C07321=1112.756,31.841,-53.401,179.866,6.990,149.335
C07322=1112.751,32.090,-53.417,179.867,6.994,149.335
C07323=1112.747,32.340,-53.432,179.868,6.998,149.336
C07324=1112.742,32.589,-53.448,179.869,7.003,149.337
C07325=1112.736,32.839,-53.464,179.870,7.007,149.337
C07326=1112.731,33.089,-53.480,179.870,7.011,149.338
C07327=1112.727,33.338,-53.495,179.871,7.015,149.339
C07328=1112.722,33.587,-53.511,179.872,7.020,149.339
C07329=1112.717,33.837,-53.527,179.874,7.024,149.340
C07330=1112.711,34.086,-53.542,179.875,7.028,149.341
C07331=1112.706,34.336,-53.558,179.875,7.032,149.341
C07332=1112.702,34.585,-53.573,179.876,7.036,149.342
C07333=1112.697,34.834,-53.590,179.877,7.040,149.343
C07334=1112.692,35.084,-53.605,179.878,7.045,149.343
C07335=1112.687,35.334,-53.621,179.879,7.049,149.344
C07336=1112.681,35.583,-53.637,179.880,7.053,149.345
C07337=1112.676,35.832,-53.653,179.881,7.057,149.345
C07338=1112.672,36.046,-53.667,179.882,7.061,149.346
C07339=1112.668,36.260,-53.680,179.883,7.064,149.346
C07340=1112.664,36.475,-53.693,179.884,7.067,149.347
C07341=1112.660,36.690,-53.707,179.884,7.071,149.348
C07342=1112.655,36.904,-53.720,179.885,7.075,149.348
C07343=1112.651,37.118,-53.734,179.886,7.078,149.349
C07344=1112.647,37.332,-53.748,179.887,7.082,149.349
C07345=1112.642,37.547,-53.761,179.888,7.086,149.350
C07346=1112.637,37.796,-53.778,179.889,7.089,149.350
C07347=1112.633,38.046,-53.794,179.890,7.094,149.351
C07348=1112.627,38.294,-53.810,179.891,7.098,149.352
C07349=1112.622,38.544,-53.826,179.892,7.102,149.352
C07350=1112.617,38.794,-53.842,179.893,7.107,149.353
C07351=1112.612,39.043,-53.858,179.893,7.110,149.354
C07352=1112.607,39.293,-53.874,179.895,7.114,149.354
C07353=1112.602,39.542,-53.890,179.896,7.118,149.355
C07354=1112.598,39.792,-53.906,179.897,7.123,149.355
C07355=1112.592,40.041,-53.922,179.898,7.127,149.356
C07356=1112.588,40.290,-53.938,179.899,7.130,149.357
C07357=1112.583,40.540,-53.953,179.900,7.135,149.357
C07358=1112.578,40.789,-53.970,179.901,7.139,149.358
C07359=1112.573,41.039,-53.986,179.902,7.143,149.359
C07360=1112.568,41.287,-54.002,179.903,7.147,149.359
C07361=1112.563,41.538,-54.018,179.904,7.152,149.360
C07362=1112.557,41.787,-54.035,179.905,7.155,149.360
C07363=1112.553,42.037,-54.051,179.906,7.159,149.361
C07364=1112.548,42.285,-54.067,179.907,7.164,149.362
C07365=1112.543,42.536,-54.083,179.908,7.168,149.362
C07366=1112.538,42.784,-54.099,179.910,7.172,149.363
C07367=1112.533,43.034,-54.115,179.910,7.175,149.363
C07368=1112.528,43.283,-54.131,179.911,7.180,149.364
C07369=1112.523,43.533,-54.147,179.912,7.184,149.365
C07370=1112.518,43.782,-54.164,179.913,7.188,149.365
C07371=1112.514,44.032,-54.180,179.915,7.192,149.366
C07372=1112.508,44.281,-54.196,179.915,7.196,149.366
C07373=1112.504,44.531,-54.213,179.916,7.200,149.367
C07374=1112.499,44.779,-54.229,179.917,7.204,149.368
C07375=1112.494,45.029,-54.245,179.919,7.208,149.368
C07376=1112.489,45.278,-54.261,179.920,7.213,149.369
C07377=1112.483,45.529,-54.278,179.921,7.217,149.369
C07378=1112.479,45.778,-54.294,179.922,7.220,149.370
C07379=1112.474,46.027,-54.311,179.923,7.224,149.371
C07380=1112.469,46.277,-54.327,179.924,7.229,149.371
C07381=1112.464,46.526,-54.343,179.925,7.233,149.372
C07382=1112.459,46.775,-54.360,179.927,7.237,149.372
C07383=1112.454,47.024,-54.376,179.927,7.240,149.373
C07384=1112.449,47.274,-54.393,179.928,7.245,149.374
C07385=1112.444,47.524,-54.409,179.929,7.249,149.374
C07386=1112.439,47.773,-54.425,179.931,7.253,149.375
C07387=1112.435,48.022,-54.442,179.932,7.257,149.375
C07388=1112.429,48.272,-54.458,179.933,7.261,149.376
C07389=1112.424,48.521,-54.475,179.934,7.265,149.376
C07390=1112.420,48.771,-54.492,179.935,7.269,149.377
C07391=1112.414,49.020,-54.508,179.936,7.273,149.378
C07392=1112.410,49.269,-54.525,179.938,7.277,149.378
C07393=1112.405,49.519,-54.540,179.939,7.281,149.379
C07394=1112.400,49.733,-54.556,179.940,7.284,149.379
C07395=1112.396,49.948,-54.569,179.940,7.288,149.380
C07396=1112.392,50.161,-54.584,179.942,7.292,149.380
C07397=1112.388,50.376,-54.597,179.943,7.295,149.381
C07398=1112.384,50.589,-54.612,179.944,7.298,149.381
C07399=1112.379,50.804,-54.626,179.944,7.302,149.382
C07400=1112.375,51.018,-54.641,179.946,7.306,149.382
C07401=1112.371,51.233,-54.655,179.947,7.309,149.383
C07402=1112.366,51.481,-54.671,179.948,7.313,149.383
C07403=1112.361,51.731,-54.688,179.949,7.317,149.384
C07404=1112.356,51.981,-54.705,179.950,7.320,149.384
C07405=1112.351,52.230,-54.721,179.951,7.325,149.385
C07406=1112.346,52.479,-54.738,179.952,7.329,149.386
C07407=1112.342,52.729,-54.755,179.954,7.333,149.386
C07408=1112.337,52.978,-54.771,179.955,7.337,149.387
C07409=1112.331,53.227,-54.789,179.956,7.341,149.387
C07410=1112.327,53.477,-54.805,179.957,7.344,149.388
C07411=1112.322,53.726,-54.822,179.958,7.349,149.388
C07412=1112.317,53.975,-54.839,179.959,7.353,149.389
C07413=1112.312,54.225,-54.856,179.961,7.357,149.389
C07414=1112.306,54.474,-54.873,179.962,7.361,149.390
C07415=1112.302,54.724,-54.889,179.964,7.365,149.391
C07416=1112.297,54.973,-54.906,179.964,7.368,149.391
C07417=1112.292,55.223,-54.923,179.966,7.372,149.392
C07418=1112.287,55.472,-54.939,179.967,7.377,149.392
C07419=1112.282,55.721,-54.957,179.968,7.381,149.393
C07420=1112.277,55.971,-54.973,179.969,7.385,149.393
C07421=1112.272,56.220,-54.990,179.970,7.389,149.394
C07422=1112.267,56.469,-55.007,179.971,7.392,149.394
C07423=1112.263,56.719,-55.024,179.972,7.397,149.395
C07424=1112.257,56.969,-55.041,179.974,7.401,149.396
C07425=1112.253,57.217,-55.058,179.975,7.405,149.396
C07426=1112.247,57.467,-55.075,179.977,7.409,149.397
C07427=1112.243,57.716,-55.092,179.978,7.413,149.397
C07428=1112.238,57.966,-55.109,179.979,7.416,149.398
C07429=1112.233,58.215,-55.126,179.980,7.420,149.398
C07430=1112.227,58.465,-55.143,179.981,7.424,149.399
C07431=1112.223,58.713,-55.160,179.982,7.429,149.399
C07432=1112.218,58.963,-55.177,179.984,7.433,149.400
C07433=1112.213,59.213,-55.194,179.985,7.437,149.400
C07434=1112.208,59.462,-55.211,179.987,7.441,149.401
C07435=1112.203,59.711,-55.228,179.988,7.444,149.401
C07436=1112.198,59.960,-55.246,179.989,7.448,149.402
C07437=1112.194,60.210,-55.262,179.990,7.452,149.402
C07438=1112.189,60.460,-55.279,179.991,7.456,149.403
C07439=1112.184,60.709,-55.297,179.993,7.460,149.404
C07440=1112.179,60.958,-55.314,179.994,7.465,149.404
C07441=1112.174,61.207,-55.330,179.995,7.468,149.405
C07442=1112.169,61.456,-55.348,179.996,7.472,149.405
C07443=1112.164,61.706,-55.366,179.998,7.476,149.406
C07444=1112.159,61.956,-55.382,179.999,7.480,149.406
C07445=1112.155,62.205,-55.400,-180.000,7.484,149.407
C07446=1112.150,62.454,-55.417,-179.998,7.488,149.407
C07447=1112.145,62.704,-55.434,-179.997,7.492,149.408
C07448=1112.139,62.953,-55.452,-179.996,7.495,149.408
C07449=1112.135,63.202,-55.469,-179.995,7.500,149.409
C07450=1112.131,63.417,-55.484,-179.993,7.504,149.409
C07451=1112.127,63.630,-55.498,-179.993,7.507,149.410
C07452=1112.122,63.844,-55.513,-179.992,7.510,149.410
C07453=1112.119,64.059,-55.528,-179.990,7.514,149.411
C07454=1112.114,64.273,-55.543,-179.989,7.517,149.411
C07455=1112.109,64.487,-55.558,-179.988,7.520,149.412
C07456=1112.106,64.701,-55.573,-179.987,7.524,149.412
C07457=1112.101,64.915,-55.588,-179.986,7.527,149.412
C07458=1112.097,65.164,-55.605,-179.984,7.531,149.413
C07459=1112.092,65.414,-55.623,-179.983,7.535,149.413
C07460=1112.087,65.663,-55.641,-179.981,7.539,149.414
C07461=1112.082,65.913,-55.657,-179.981,7.543,149.415
C07462=1112.077,66.162,-55.675,-179.979,7.547,149.415
C07463=1112.072,66.412,-55.693,-179.978,7.550,149.415
C07464=1112.067,66.660,-55.710,-179.977,7.555,149.416
C07465=1112.062,66.910,-55.727,-179.975,7.559,149.417
C07466=1112.057,67.159,-55.745,-179.974,7.563,149.417
C07467=1112.052,67.409,-55.762,-179.972,7.567,149.418
C07468=1112.048,67.657,-55.779,-179.971,7.571,149.418
C07469=1112.043,67.907,-55.797,-179.970,7.574,149.419
C07470=1112.038,68.156,-55.815,-179.969,7.578,149.419
C07471=1112.033,68.406,-55.833,-179.967,7.582,149.420
C07472=1112.028,68.655,-55.850,-179.966,7.586,149.420
C07473=1112.023,68.904,-55.867,-179.964,7.590,149.421
C07474=1112.018,69.153,-55.885,-179.963,7.594,149.421
C07475=1112.013,69.403,-55.903,-179.962,7.598,149.422
C07476=1112.008,69.652,-55.921,-179.960,7.602,149.422
C07477=1112.003,69.902,-55.938,-179.959,7.606,149.423
C07478=1111.999,70.151,-55.955,-179.958,7.610,149.423
C07479=1111.994,70.400,-55.973,-179.957,7.614,149.424
C07480=1111.989,70.649,-55.991,-179.955,7.618,149.424
C07481=1111.984,70.899,-56.008,-179.954,7.622,149.425
C07482=1111.979,71.148,-56.026,-179.952,7.626,149.425
C07483=1111.974,71.397,-56.044,-179.951,7.630,149.426
C07484=1111.969,71.647,-56.062,-179.949,7.634,149.426
C07485=1111.965,71.896,-56.079,-179.948,7.638,149.427
C07486=1111.960,72.146,-56.097,-179.947,7.642,149.427
C07487=1111.955,72.395,-56.115,-179.945,7.646,149.428
C07488=1111.951,72.644,-56.133,-179.944,7.649,149.428
C07489=1111.945,72.894,-56.151,-179.943,7.653,149.429
C07490=1111.940,73.143,-56.169,-179.941,7.657,149.429
C07491=1111.936,73.393,-56.187,-179.940,7.661,149.430
C07492=1111.931,73.642,-56.205,-179.939,7.665,149.430
C07493=1111.926,73.891,-56.222,-179.937,7.669,149.431
C07494=1111.921,74.140,-56.240,-179.935,7.673,149.431
C07495=1111.916,74.389,-56.258,-179.934,7.677,149.432
C07496=1111.911,74.639,-56.276,-179.933,7.681,149.432
C07497=1111.906,74.888,-56.294,-179.931,7.685,149.433
C07498=1111.901,75.138,-56.312,-179.930,7.689,149.433
C07499=1111.897,75.387,-56.330,-179.928,7.693,149.434
C07500=1111.892,75.636,-56.348,-179.928,7.696,149.434
C07501=1111.887,75.886,-56.366,-179.926,7.700,149.434
C07502=1111.882,76.135,-56.384,-179.925,7.704,149.435
C07503=1111.877,76.384,-56.402,-179.923,7.708,149.436
C07504=1111.872,76.633,-56.420,-179.922,7.712,149.436
C07505=1111.867,76.882,-56.438,-179.920,7.716,149.436
C07506=1111.864,77.097,-56.453,-179.920,7.720,149.437
C07507=1111.859,77.310,-56.468,-179.919,7.723,149.438
C07508=1111.855,77.525,-56.484,-179.918,7.726,149.438
C07509=1111.851,77.738,-56.500,-179.917,7.729,149.438
C07510=1111.847,77.953,-56.515,-179.916,7.732,149.439
C07511=1111.843,78.167,-56.531,-179.915,7.736,149.439
C07512=1111.838,78.380,-56.547,-179.914,7.739,149.440
C07513=1111.834,78.595,-56.562,-179.913,7.742,149.440
C07514=1111.829,78.844,-56.580,-179.913,7.745,149.441
C07515=1111.824,79.094,-56.598,-179.911,7.749,149.441
C07516=1111.819,79.343,-56.616,-179.911,7.753,149.442
C07517=1111.815,79.592,-56.634,-179.909,7.757,149.442
C07518=1111.810,79.841,-56.652,-179.909,7.760,149.443
C07519=1111.806,80.090,-56.671,-179.907,7.764,149.444
C07520=1111.801,80.339,-56.689,-179.907,7.768,149.444
C07521=1111.795,80.589,-56.708,-179.905,7.771,149.445
C07522=1111.790,80.838,-56.726,-179.904,7.775,149.445
C07523=1111.786,81.088,-56.744,-179.903,7.779,149.446
C07524=1111.781,81.337,-56.762,-179.902,7.783,149.446
C07525=1111.776,81.586,-56.780,-179.901,7.787,149.447
C07526=1111.771,81.836,-56.798,-179.900,7.790,149.447
C07527=1111.767,82.084,-56.817,-179.899,7.794,149.448
C07528=1111.761,82.334,-56.836,-179.898,7.798,149.449
C07529=1111.757,82.583,-56.854,-179.897,7.801,149.449
C07530=1111.752,82.833,-56.872,-179.895,7.805,149.450
C07531=1111.747,83.082,-56.889,-179.894,7.809,149.450
C07532=1111.743,83.331,-56.909,-179.893,7.813,149.451
C07533=1111.737,83.581,-56.927,-179.892,7.817,149.451
C07534=1111.732,83.830,-56.945,-179.891,7.820,149.452
C07535=1111.727,84.079,-56.963,-179.890,7.824,149.452
C07536=1111.723,84.328,-56.982,-179.889,7.828,149.453
C07537=1111.718,84.577,-57.000,-179.888,7.831,149.453
C07538=1111.713,84.827,-57.019,-179.886,7.836,149.454
C07539=1111.708,85.077,-57.037,-179.885,7.839,149.454
C07540=1111.704,85.325,-57.056,-179.884,7.843,149.455
C07541=1111.699,85.574,-57.074,-179.883,7.847,149.455
C07542=1111.693,85.824,-57.092,-179.881,7.851,149.456
C07543=1111.689,86.073,-57.111,-179.881,7.854,149.457
C07544=1111.684,86.322,-57.129,-179.879,7.858,149.457
C07545=1111.679,86.572,-57.148,-179.877,7.862,149.457
C07546=1111.675,86.821,-57.167,-179.877,7.866,149.458
C07547=1111.670,87.070,-57.185,-179.875,7.869,149.458
C07548=1111.665,87.319,-57.204,-179.874,7.874,149.459
C07549=1111.660,87.569,-57.223,-179.873,7.877,149.460
C07550=1111.655,87.818,-57.241,-179.872,7.881,149.460
C07551=1111.651,88.067,-57.259,-179.871,7.885,149.461
C07552=1111.646,88.317,-57.278,-179.870,7.888,149.461
C07553=1111.641,88.565,-57.297,-179.868,7.892,149.462
C07554=1111.636,88.815,-57.315,-179.867,7.896,149.462
C07555=1111.631,89.065,-57.334,-179.865,7.900,149.463
C07556=1111.626,89.313,-57.353,-179.864,7.903,149.463
C07557=1111.621,89.563,-57.371,-179.863,7.907,149.463
C07558=1111.617,89.812,-57.390,-179.862,7.911,149.464
C07559=1111.612,90.061,-57.408,-179.860,7.915,149.465
C07560=1111.607,90.311,-57.428,-179.859,7.918,149.465
C07561=1111.602,90.560,-57.446,-179.857,7.922,149.465
C07562=1111.598,90.774,-57.462,-179.856,7.925,149.466
C07563=1111.594,90.988,-57.478,-179.855,7.929,149.466
C07564=1111.589,91.202,-57.494,-179.854,7.932,149.467
C07565=1111.586,91.415,-57.511,-179.853,7.936,149.467
C07566=1111.581,91.629,-57.527,-179.852,7.939,149.468
C07567=1111.578,91.843,-57.543,-179.850,7.943,149.468
C07568=1111.574,92.057,-57.559,-179.849,7.946,149.468
C07569=1111.570,92.271,-57.575,-179.848,7.949,149.469
C07570=1111.564,92.521,-57.594,-179.847,7.953,149.469
C07571=1111.560,92.769,-57.612,-179.845,7.957,149.470
C07572=1111.555,93.019,-57.632,-179.844,7.960,149.470
C07573=1111.550,93.268,-57.650,-179.843,7.964,149.471
C07574=1111.545,93.517,-57.670,-179.841,7.967,149.471
C07575=1111.540,93.767,-57.688,-179.840,7.972,149.472
C07576=1111.536,94.016,-57.707,-179.838,7.976,149.472
C07577=1111.531,94.265,-57.726,-179.837,7.979,149.473
C07578=1111.525,94.514,-57.745,-179.835,7.983,149.473
C07579=1111.521,94.764,-57.764,-179.834,7.986,149.473
C07580=1111.516,95.012,-57.783,-179.833,7.990,149.474
C07581=1111.512,95.262,-57.802,-179.831,7.994,149.474
C07582=1111.506,95.511,-57.821,-179.829,7.998,149.475
C07583=1111.502,95.761,-57.840,-179.828,8.002,149.475
C07584=1111.497,96.009,-57.859,-179.826,8.006,149.476
C07585=1111.492,96.259,-57.879,-179.825,8.010,149.476
C07586=1111.487,96.508,-57.897,-179.824,8.013,149.476
C07587=1111.483,96.758,-57.916,-179.822,8.017,149.477
C07588=1111.478,97.006,-57.935,-179.820,8.021,149.477
C07589=1111.473,97.256,-57.955,-179.819,8.025,149.478
C07590=1111.468,97.505,-57.973,-179.817,8.028,149.478
C07591=1111.464,97.754,-57.992,-179.816,8.032,149.479
C07592=1111.458,98.003,-58.012,-179.814,8.036,149.479
C07593=1111.454,98.253,-58.031,-179.812,8.040,149.480
C07594=1111.450,98.502,-58.050,-179.811,8.044,149.480
C07595=1111.444,98.751,-58.070,-179.809,8.048,149.480
C07596=1111.440,99.000,-58.089,-179.808,8.051,149.481
C07597=1111.435,99.249,-58.108,-179.807,8.055,149.481
C07598=1111.430,99.499,-58.127,-179.805,8.059,149.482
C07599=1111.425,99.748,-58.146,-179.803,8.062,149.482
C07600=1111.420,99.997,-58.165,-179.801,8.066,149.482
C07601=1111.415,100.246,-58.184,-179.800,8.070,149.483
C07602=1111.411,100.496,-58.204,-179.798,8.074,149.483
C07603=1111.406,100.745,-58.223,-179.796,8.078,149.484
C07604=1111.401,100.994,-58.242,-179.794,8.081,149.484
C07605=1111.396,101.244,-58.262,-179.793,8.085,149.484
C07606=1111.392,101.492,-58.281,-179.791,8.089,149.485
C07607=1111.387,101.742,-58.300,-179.790,8.093,149.485
C07608=1111.382,101.991,-58.320,-179.788,8.097,149.486
C07609=1111.377,102.240,-58.339,-179.786,8.100,149.486
C07610=1111.373,102.489,-58.358,-179.784,8.104,149.486
C07611=1111.367,102.738,-58.378,-179.783,8.108,149.487
C07612=1111.363,102.988,-58.397,-179.781,8.112,149.487
C07613=1111.358,103.237,-58.417,-179.779,8.116,149.487
C07614=1111.353,103.486,-58.436,-179.777,8.119,149.488
C07615=1111.349,103.735,-58.456,-179.775,8.123,149.488
C07616=1111.344,103.984,-58.476,-179.774,8.127,149.488
C07617=1111.339,104.233,-58.495,-179.772,8.131,149.489
C07618=1111.335,104.447,-58.511,-179.771,8.133,149.489
C07619=1111.331,104.661,-58.529,-179.769,8.137,149.489
C07620=1111.327,104.875,-58.545,-179.768,8.140,149.490
C07621=1111.323,105.089,-58.562,-179.766,8.143,149.490
C07622=1111.319,105.303,-58.579,-179.764,8.146,149.490
C07623=1111.315,105.517,-58.596,-179.763,8.149,149.491
C07624=1111.311,105.730,-58.612,-179.761,8.153,149.491
C07625=1111.306,105.944,-58.629,-179.760,8.156,149.491
C07626=1111.302,106.193,-58.649,-179.758,8.159,149.492
C07627=1111.297,106.443,-58.669,-179.756,8.163,149.492
C07628=1111.292,106.692,-58.688,-179.755,8.167,149.492
C07629=1111.287,106.941,-58.708,-179.752,8.170,149.492
C07630=1111.283,107.190,-58.728,-179.751,8.174,149.493
C07631=1111.278,107.439,-58.747,-179.749,8.178,149.493
C07632=1111.273,107.688,-58.766,-179.747,8.181,149.493
C07633=1111.268,107.937,-58.787,-179.745,8.185,149.494
C07634=1111.264,108.187,-58.807,-179.742,8.189,149.494
C07635=1111.259,108.436,-58.826,-179.740,8.193,149.494
C07636=1111.254,108.685,-58.845,-179.739,8.197,149.495
C07637=1111.249,108.934,-58.866,-179.737,8.200,149.495
C07638=1111.244,109.184,-58.885,-179.735,8.204,149.495
C07639=1111.240,109.433,-58.906,-179.733,8.208,149.496
C07640=1111.235,109.681,-58.925,-179.731,8.211,149.496
C07641=1111.230,109.931,-58.945,-179.729,8.215,149.496
C07642=1111.226,110.180,-58.965,-179.727,8.218,149.496
C07643=1111.221,110.430,-58.985,-179.725,8.222,149.497
C07644=1111.216,110.679,-59.005,-179.723,8.226,149.497
C07645=1111.211,110.927,-59.024,-179.721,8.229,149.497
C07646=1111.206,111.177,-59.044,-179.719,8.233,149.497
C07647=1111.202,111.426,-59.065,-179.717,8.236,149.498
C07648=1111.197,111.675,-59.084,-179.715,8.240,149.498
C07649=1111.193,111.924,-59.105,-179.713,8.243,149.498
C07650=1111.187,112.173,-59.124,-179.712,8.247,149.499
C07651=1111.183,112.422,-59.144,-179.710,8.250,149.499
C07652=1111.177,112.672,-59.164,-179.708,8.254,149.499
C07653=1111.173,112.921,-59.185,-179.707,8.257,149.500
C07654=1111.168,113.170,-59.205,-179.705,8.260,149.500
C07655=1111.164,113.420,-59.225,-179.704,8.264,149.500
C07656=1111.159,113.668,-59.245,-179.702,8.268,149.500
C07657=1111.154,113.917,-59.265,-179.699,8.271,149.501
C07658=1111.150,114.166,-59.285,-179.698,8.274,149.501
C07659=1111.145,114.416,-59.305,-179.696,8.278,149.501
C07660=1111.140,114.665,-59.326,-179.694,8.281,149.502
C07661=1111.135,114.914,-59.346,-179.693,8.284,149.502
C07662=1111.130,115.164,-59.366,-179.691,8.288,149.502
C07663=1111.125,115.412,-59.386,-179.689,8.291,149.502
C07664=1111.121,115.661,-59.406,-179.687,8.295,149.503
C07665=1111.116,115.910,-59.426,-179.686,8.298,149.503
C07666=1111.111,116.160,-59.447,-179.684,8.301,149.503
C07667=1111.107,116.409,-59.467,-179.682,8.305,149.504
C07668=1111.102,116.658,-59.487,-179.680,8.309,149.504
C07669=1111.097,116.907,-59.507,-179.679,8.311,149.504
C07670=1111.093,117.156,-59.527,-179.677,8.315,149.504
C07671=1111.088,117.405,-59.548,-179.675,8.318,149.505
C07672=1111.083,117.655,-59.568,-179.673,8.322,149.505
C07673=1111.079,117.904,-59.588,-179.672,8.325,149.505
C07674=1111.074,118.118,-59.606,-179.670,8.328,149.506
C07675=1111.070,118.331,-59.623,-179.668,8.331,149.506
C07676=1111.066,118.545,-59.641,-179.667,8.334,149.506
C07677=1111.062,118.758,-59.659,-179.665,8.337,149.506
C07678=1111.058,118.972,-59.676,-179.664,8.339,149.506
C07679=1111.054,119.186,-59.693,-179.663,8.342,149.507
C07680=1111.050,119.399,-59.710,-179.661,8.346,149.507
C07681=1111.046,119.613,-59.728,-179.660,8.349,149.507
C07682=1111.041,119.862,-59.748,-179.658,8.351,149.508
C07683=1111.036,120.111,-59.769,-179.656,8.355,149.508
C07684=1111.032,120.360,-59.789,-179.654,8.358,149.508
C07685=1111.027,120.609,-59.810,-179.652,8.362,149.508
C07686=1111.022,120.859,-59.831,-179.651,8.365,149.509
C07687=1111.017,121.108,-59.850,-179.649,8.369,149.509
C07688=1111.013,121.357,-59.871,-179.647,8.372,149.509
C07689=1111.008,121.606,-59.892,-179.646,8.375,149.510
C07690=1111.003,121.855,-59.912,-179.644,8.379,149.510
C07691=1110.999,122.104,-59.933,-179.642,8.382,149.510
C07692=1110.994,122.354,-59.953,-179.640,8.385,149.510
C07693=1110.989,122.602,-59.974,-179.639,8.389,149.511
C07694=1110.984,122.852,-59.995,-179.637,8.392,149.511
C07695=1110.980,123.101,-60.015,-179.635,8.395,149.511
C07696=1110.975,123.350,-60.036,-179.633,8.398,149.511
C07697=1110.970,123.599,-60.057,-179.631,8.402,149.512
C07698=1110.966,123.849,-60.077,-179.629,8.406,149.512
C07699=1110.961,124.098,-60.098,-179.628,8.409,149.512
C07700=1110.956,124.347,-60.119,-179.626,8.412,149.512
C07701=1110.952,124.596,-60.139,-179.624,8.416,149.513
C07702=1110.947,124.845,-60.160,-179.623,8.419,149.513
C07703=1110.942,125.094,-60.180,-179.621,8.422,149.513
C07704=1110.937,125.343,-60.201,-179.619,8.426,149.514
C07705=1110.933,125.592,-60.222,-179.618,8.429,149.514
C07706=1110.928,125.841,-60.243,-179.616,8.432,149.514
C07707=1110.924,126.090,-60.264,-179.614,8.436,149.514
C07708=1110.918,126.339,-60.285,-179.612,8.438,149.515
C07709=1110.914,126.588,-60.305,-179.610,8.442,149.515
C07710=1110.909,126.838,-60.326,-179.608,8.446,149.515
C07711=1110.905,127.087,-60.347,-179.607,8.449,149.516
C07712=1110.900,127.335,-60.368,-179.605,8.452,149.516
C07713=1110.896,127.584,-60.389,-179.603,8.456,149.516
C07714=1110.890,127.834,-60.410,-179.602,8.459,149.517
C07715=1110.886,128.083,-60.430,-179.600,8.462,149.517
C07716=1110.881,128.332,-60.451,-179.598,8.466,149.517
C07717=1110.876,128.581,-60.473,-179.596,8.468,149.517
C07718=1110.872,128.830,-60.494,-179.595,8.472,149.518
C07719=1110.867,129.079,-60.514,-179.593,8.476,149.518
C07720=1110.862,129.328,-60.535,-179.591,8.479,149.518
C07721=1110.858,129.577,-60.557,-179.589,8.482,149.518
C07722=1110.853,129.826,-60.577,-179.587,8.486,149.519
C07723=1110.848,130.075,-60.598,-179.585,8.489,149.519
C07724=1110.843,130.324,-60.620,-179.584,8.492,149.519
C07725=1110.839,130.574,-60.640,-179.582,8.495,149.519
C07726=1110.834,130.823,-60.661,-179.580,8.499,149.520
C07727=1110.829,131.071,-60.683,-179.579,8.502,149.520
C07728=1110.825,131.320,-60.703,-179.577,8.506,149.520
C07729=1110.820,131.570,-60.724,-179.575,8.509,149.521
C07730=1110.816,131.784,-60.743,-179.574,8.512,149.521
C07731=1110.812,131.997,-60.761,-179.572,8.515,149.521
C07732=1110.808,132.210,-60.778,-179.571,8.518,149.521
C07733=1110.803,132.424,-60.797,-179.569,8.520,149.522
C07734=1110.800,132.638,-60.816,-179.568,8.523,149.522
C07735=1110.796,132.852,-60.833,-179.566,8.526,149.522
C07736=1110.792,133.065,-60.851,-179.564,8.529,149.522
C07737=1110.788,133.279,-60.870,-179.563,8.532,149.523
C07738=1110.783,133.528,-60.891,-179.562,8.535,149.523
C07739=1110.778,133.777,-60.912,-179.560,8.539,149.523
C07740=1110.773,134.026,-60.933,-179.558,8.542,149.524
C07741=1110.770,134.275,-60.955,-179.556,8.545,149.524
C07742=1110.765,134.524,-60.976,-179.555,8.549,149.524
C07743=1110.760,134.773,-60.997,-179.553,8.552,149.524
C07744=1110.755,135.022,-61.018,-179.551,8.556,149.525
C07745=1110.751,135.271,-61.040,-179.550,8.559,149.525
C07746=1110.746,135.520,-61.061,-179.547,8.562,149.525
C07747=1110.741,135.769,-61.082,-179.545,8.566,149.526
C07748=1110.736,136.018,-61.103,-179.544,8.569,149.526
C07749=1110.732,136.268,-61.125,-179.542,8.572,149.526
C07750=1110.727,136.516,-61.146,-179.540,8.576,149.526
C07751=1110.722,136.765,-61.167,-179.539,8.579,149.527
C07752=1110.718,137.014,-61.189,-179.537,8.582,149.527
C07753=1110.713,137.264,-61.210,-179.535,8.586,149.527
C07754=1110.708,137.512,-61.232,-179.534,8.589,149.528
C07755=1110.704,137.761,-61.254,-179.532,8.592,149.528
C07756=1110.699,138.011,-61.275,-179.530,8.596,149.528
C07757=1110.694,138.259,-61.296,-179.529,8.599,149.529
C07758=1110.690,138.509,-61.318,-179.527,8.602,149.529
C07759=1110.685,138.758,-61.339,-179.525,8.606,149.529
C07760=1110.680,139.007,-61.361,-179.524,8.609,149.530
C07761=1110.676,139.256,-61.383,-179.522,8.613,149.530
C07762=1110.671,139.505,-61.403,-179.520,8.616,149.530
C07763=1110.666,139.753,-61.425,-179.519,8.619,149.530
C07764=1110.662,140.003,-61.447,-179.517,8.623,149.531
C07765=1110.657,140.251,-61.469,-179.515,8.626,149.531
C07766=1110.652,140.501,-61.490,-179.513,8.630,149.531
C07767=1110.648,140.750,-61.512,-179.511,8.633,149.532
C07768=1110.643,140.999,-61.533,-179.510,8.637,149.532
C07769=1110.639,141.248,-61.556,-179.508,8.640,149.532
C07770=1110.634,141.497,-61.576,-179.507,8.643,149.533
C07771=1110.629,141.746,-61.598,-179.505,8.647,149.533
C07772=1110.624,141.995,-61.620,-179.503,8.650,149.533
C07773=1110.620,142.244,-61.642,-179.502,8.653,149.534
C07774=1110.615,142.493,-61.664,-179.499,8.657,149.534
C07775=1110.611,142.742,-61.685,-179.498,8.661,149.534
C07776=1110.606,142.991,-61.706,-179.496,8.664,149.535
C07777=1110.602,143.240,-61.728,-179.495,8.667,149.535
C07778=1110.597,143.489,-61.750,-179.493,8.671,149.535
C07779=1110.593,143.738,-61.772,-179.491,8.674,149.536
C07780=1110.588,143.987,-61.793,-179.490,8.677,149.536
C07781=1110.583,144.236,-61.815,-179.488,8.681,149.536
C07782=1110.578,144.485,-61.838,-179.486,8.685,149.537
C07783=1110.573,144.734,-61.859,-179.485,8.688,149.537
C07784=1110.569,144.983,-61.882,-179.483,8.691,149.537
C07785=1110.564,145.232,-61.903,-179.481,8.695,149.538
C07786=1110.560,145.446,-61.922,-179.480,8.698,149.538
C07787=1110.556,145.659,-61.940,-179.478,8.701,149.538
C07788=1110.552,145.873,-61.959,-179.476,8.704,149.538
C07789=1110.548,146.086,-61.978,-179.474,8.707,149.539
C07790=1110.545,146.300,-61.997,-179.473,8.710,149.539
C07791=1110.540,146.513,-62.016,-179.471,8.714,149.539
C07792=1110.537,146.727,-62.034,-179.469,8.716,149.539
C07793=1110.532,146.940,-62.053,-179.467,8.720,149.540
C07794=1110.528,147.189,-62.076,-179.465,8.723,149.540
C07795=1110.523,147.438,-62.097,-179.463,8.727,149.540
C07796=1110.519,147.687,-62.119,-179.461,8.730,149.540
C07797=1110.514,147.936,-62.141,-179.459,8.734,149.541
C07798=1110.509,148.185,-62.164,-179.457,8.738,149.541
C07799=1110.504,148.434,-62.185,-179.455,8.741,149.541
C07800=1110.500,148.683,-62.207,-179.453,8.745,149.541
C07801=1110.495,148.931,-62.230,-179.451,8.748,149.542
C07802=1110.491,149.181,-62.252,-179.449,8.752,149.542
C07803=1110.485,149.430,-62.274,-179.447,8.755,149.542
C07804=1110.481,149.679,-62.296,-179.445,8.759,149.542
C07805=1110.476,149.928,-62.318,-179.442,8.762,149.543
C07806=1110.472,150.177,-62.340,-179.440,8.766,149.543
C07807=1110.468,150.426,-62.363,-179.438,8.769,149.543
C07808=1110.463,150.675,-62.385,-179.436,8.773,149.543
C07809=1110.458,150.924,-62.407,-179.435,8.775,149.544
C07810=1110.453,151.173,-62.429,-179.433,8.779,149.544
C07811=1110.449,151.421,-62.451,-179.431,8.782,149.544
C07812=1110.444,151.670,-62.474,-179.429,8.786,149.544
C07813=1110.440,151.920,-62.496,-179.426,8.789,149.544
C07814=1110.435,152.169,-62.518,-179.424,8.793,149.545
C07815=1110.430,152.417,-62.541,-179.422,8.796,149.545
C07816=1110.426,152.667,-62.563,-179.420,8.799,149.545
C07817=1110.421,152.915,-62.584,-179.418,8.803,149.545
C07818=1110.416,153.164,-62.608,-179.416,8.806,149.545
C07819=1110.412,153.414,-62.630,-179.414,8.810,149.546
C07820=1110.407,153.662,-62.652,-179.411,8.813,149.546
C07821=1110.402,153.911,-62.675,-179.410,8.816,149.546
C07822=1110.398,154.161,-62.697,-179.407,8.819,149.546
C07823=1110.393,154.409,-62.719,-179.405,8.823,149.546
C07824=1110.388,154.658,-62.742,-179.403,8.826,149.547
C07825=1110.385,154.907,-62.765,-179.401,8.829,149.547
C07826=1110.380,155.156,-62.786,-179.399,8.833,149.547
C07827=1110.375,155.405,-62.809,-179.397,8.836,149.547
C07828=1110.371,155.654,-62.832,-179.395,8.840,149.547
C07829=1110.365,155.903,-62.854,-179.393,8.842,149.548
C07830=1110.361,156.152,-62.877,-179.391,8.845,149.548
C07831=1110.357,156.401,-62.899,-179.389,8.849,149.548
C07832=1110.352,156.650,-62.922,-179.386,8.852,149.548
C07833=1110.347,156.899,-62.944,-179.384,8.855,149.548
C07834=1110.343,157.148,-62.967,-179.382,8.859,149.548
C07835=1110.338,157.396,-62.990,-179.380,8.862,149.549
C07836=1110.333,157.646,-63.012,-179.378,8.865,149.549
C07837=1110.329,157.894,-63.035,-179.376,8.868,149.549
C07838=1110.325,158.144,-63.057,-179.374,8.872,149.549
C07839=1110.319,158.392,-63.080,-179.371,8.875,149.549
C07840=1110.316,158.641,-63.103,-179.369,8.878,149.549
C07841=1110.310,158.890,-63.126,-179.368,8.881,149.550
C07842=1110.306,159.103,-63.145,-179.365,8.884,149.550
C07843=1110.302,159.317,-63.165,-179.364,8.887,149.550
C07844=1110.299,159.530,-63.185,-179.362,8.889,149.550
C07845=1110.295,159.743,-63.203,-179.360,8.892,149.550
C07846=1110.291,159.957,-63.223,-179.358,8.895,149.550
C07847=1110.287,160.171,-63.242,-179.356,8.898,149.550
C07848=1110.283,160.384,-63.262,-179.354,8.900,149.551
C07849=1110.279,160.597,-63.282,-179.353,8.903,149.551
C07850=1110.274,160.846,-63.305,-179.350,8.906,149.551
C07851=1110.270,161.095,-63.327,-179.348,8.909,149.551
C07852=1110.265,161.344,-63.350,-179.346,8.912,149.551
C07853=1110.261,161.592,-63.373,-179.344,8.916,149.551
C07854=1110.256,161.841,-63.396,-179.342,8.918,149.551
C07855=1110.251,162.091,-63.419,-179.340,8.922,149.552
C07856=1110.247,162.340,-63.442,-179.337,8.925,149.552
C07857=1110.242,162.589,-63.465,-179.335,8.928,149.552
C07858=1110.238,162.838,-63.488,-179.333,8.931,149.552
C07859=1110.233,163.086,-63.511,-179.331,8.934,149.552
C07860=1110.228,163.336,-63.533,-179.329,8.937,149.552
C07861=1110.224,163.584,-63.556,-179.327,8.941,149.552
C07862=1110.219,163.833,-63.579,-179.325,8.943,149.552
C07863=1110.215,164.082,-63.603,-179.323,8.947,149.553
C07864=1110.211,164.331,-63.626,-179.320,8.950,149.553
C07865=1110.205,164.579,-63.649,-179.318,8.953,149.553
C07866=1110.201,164.828,-63.671,-179.316,8.956,149.553
C07867=1110.197,165.077,-63.695,-179.314,8.959,149.553
C07868=1110.192,165.326,-63.718,-179.312,8.962,149.553
C07869=1110.187,165.575,-63.741,-179.310,8.964,149.553
C07870=1110.183,165.824,-63.764,-179.308,8.968,149.554
C07871=1110.179,166.073,-63.787,-179.305,8.971,149.554
C07872=1110.174,166.323,-63.810,-179.303,8.975,149.554
C07873=1110.168,166.571,-63.833,-179.301,8.977,149.554
C07874=1110.164,166.820,-63.856,-179.299,8.980,149.554
C07875=1110.160,167.069,-63.879,-179.296,8.983,149.554
C07876=1110.155,167.317,-63.903,-179.295,8.986,149.554
C07877=1110.151,167.566,-63.927,-179.292,8.989,149.554
C07878=1110.147,167.815,-63.949,-179.290,8.992,149.554
C07879=1110.142,168.064,-63.973,-179.287,8.996,149.554
C07880=1110.137,168.313,-63.996,-179.286,8.998,149.555
C07881=1110.133,168.562,-64.020,-179.283,9.001,149.555
C07882=1110.128,168.811,-64.043,-179.281,9.004,149.555
C07883=1110.124,169.060,-64.066,-179.279,9.007,149.555
C07884=1110.119,169.309,-64.089,-179.277,9.010,149.555
C07885=1110.115,169.558,-64.112,-179.274,9.013,149.555
C07886=1110.109,169.806,-64.135,-179.273,9.016,149.555
C07887=1110.105,170.055,-64.159,-179.270,9.019,149.555
C07888=1110.100,170.304,-64.183,-179.268,9.023,149.556
C07889=1110.095,170.553,-64.206,-179.266,9.025,149.556
C07890=1110.091,170.801,-64.229,-179.264,9.028,149.556
C07891=1110.087,171.050,-64.252,-179.262,9.032,149.556
C07892=1110.082,171.299,-64.276,-179.260,9.034,149.556
C07893=1110.078,171.548,-64.300,-179.257,9.037,149.556
C07894=1110.073,171.797,-64.323,-179.255,9.041,149.556
C07895=1110.068,172.046,-64.346,-179.253,9.044,149.556
C07896=1110.064,172.294,-64.370,-179.251,9.046,149.556
C07897=1110.059,172.543,-64.394,-179.249,9.049,149.557
C07898=1110.055,172.757,-64.414,-179.247,9.052,149.557
C07899=1110.052,172.970,-64.434,-179.245,9.054,149.557
C07900=1110.047,173.184,-64.455,-179.243,9.056,149.557
C07901=1110.044,173.397,-64.474,-179.242,9.059,149.557
C07902=1110.040,173.610,-64.495,-179.239,9.062,149.557
C07903=1110.036,173.824,-64.515,-179.237,9.065,149.557
C07904=1110.032,174.037,-64.536,-179.235,9.067,149.557
C07905=1110.028,174.250,-64.555,-179.234,9.070,149.557
C07906=1110.023,174.499,-64.579,-179.231,9.073,149.557
C07907=1110.019,174.748,-64.603,-179.230,9.075,149.557
C07908=1110.015,174.997,-64.626,-179.227,9.079,149.558
C07909=1110.010,175.245,-64.650,-179.225,9.082,149.558
C07910=1110.006,175.494,-64.674,-179.223,9.084,149.558
C07911=1110.001,175.743,-64.698,-179.221,9.087,149.558
C07912=1109.996,175.992,-64.721,-179.218,9.091,149.558
C07913=1109.992,176.241,-64.745,-179.217,9.093,149.558
C07914=1109.987,176.489,-64.769,-179.214,9.096,149.558
C07915=1109.983,176.738,-64.792,-179.212,9.100,149.558
C07916=1109.978,176.987,-64.816,-179.210,9.102,149.558
C07917=1109.974,177.236,-64.839,-179.208,9.105,149.559
C07918=1109.970,177.485,-64.864,-179.206,9.108,149.559
C07919=1109.965,177.734,-64.887,-179.204,9.111,149.559
C07920=1109.961,177.982,-64.911,-179.201,9.114,149.559
C07921=1109.956,178.231,-64.935,-179.200,9.117,149.559
C07922=1109.951,178.480,-64.959,-179.197,9.120,149.559
C07923=1109.946,178.729,-64.983,-179.195,9.123,149.559
C07924=1109.942,178.978,-65.007,-179.193,9.126,149.559
C07925=1109.938,179.227,-65.031,-179.191,9.129,149.559
C07926=1109.933,179.476,-65.055,-179.188,9.132,149.559
C07927=1109.929,179.724,-65.079,-179.186,9.135,149.560
C07928=1109.924,179.973,-65.103,-179.184,9.138,149.560
C07929=1109.919,180.222,-65.127,-179.181,9.141,149.560
C07930=1109.915,180.470,-65.151,-179.179,9.144,149.560
C07931=1109.911,180.720,-65.175,-179.176,9.147,149.560
C07932=1109.906,180.968,-65.199,-179.174,9.150,149.560
C07933=1109.902,181.217,-65.223,-179.171,9.153,149.560
C07934=1109.897,181.465,-65.247,-179.170,9.156,149.560
C07935=1109.892,181.715,-65.271,-179.167,9.159,149.560
C07936=1109.888,181.964,-65.295,-179.165,9.162,149.560
C07937=1109.884,182.212,-65.319,-179.162,9.165,149.560
C07938=1109.879,182.461,-65.343,-179.160,9.168,149.560
C07939=1109.874,182.710,-65.367,-179.158,9.171,149.560
C07940=1109.869,182.958,-65.391,-179.155,9.174,149.560
C07941=1109.866,183.207,-65.416,-179.153,9.177,149.560
C07942=1109.861,183.456,-65.440,-179.150,9.180,149.560
C07943=1109.856,183.705,-65.464,-179.148,9.182,149.560
C07944=1109.851,183.954,-65.488,-179.146,9.185,149.560
C07945=1109.848,184.203,-65.512,-179.143,9.188,149.561
C07946=1109.843,184.451,-65.537,-179.142,9.191,149.561
C07947=1109.838,184.700,-65.561,-179.139,9.194,149.561
C07948=1109.834,184.948,-65.585,-179.137,9.197,149.561
C07949=1109.830,185.197,-65.610,-179.134,9.200,149.561
C07950=1109.825,185.447,-65.633,-179.132,9.202,149.561
C07951=1109.820,185.695,-65.658,-179.130,9.206,149.561
C07952=1109.816,185.944,-65.682,-179.127,9.209,149.561
C07953=1109.811,186.193,-65.707,-179.125,9.211,149.561
C07954=1109.808,186.406,-65.727,-179.123,9.213,149.561
C07955=1109.804,186.619,-65.748,-179.121,9.216,149.561
C07956=1109.799,186.832,-65.769,-179.119,9.219,149.561
C07957=1109.796,187.045,-65.790,-179.117,9.221,149.561
C07958=1109.792,187.259,-65.811,-179.115,9.223,149.561
C07959=1109.787,187.472,-65.832,-179.113,9.226,149.561
C07960=1109.784,187.685,-65.853,-179.111,9.228,149.561
C07961=1109.780,187.899,-65.874,-179.109,9.230,149.561
C07962=1109.776,188.147,-65.898,-179.107,9.234,149.561
C07963=1109.771,188.396,-65.923,-179.105,9.236,149.561
C07964=1109.766,188.644,-65.947,-179.102,9.239,149.561
C07965=1109.762,188.894,-65.972,-179.100,9.242,149.561
C07966=1109.758,189.142,-65.996,-179.098,9.244,149.561
C07967=1109.754,189.391,-66.021,-179.096,9.248,149.561
C07968=1109.749,189.639,-66.046,-179.094,9.250,149.561
C07969=1109.745,189.888,-66.070,-179.091,9.253,149.562
C07970=1109.740,190.137,-66.095,-179.089,9.256,149.562
C07971=1109.736,190.386,-66.119,-179.087,9.258,149.562
C07972=1109.730,190.634,-66.144,-179.084,9.262,149.562
C07973=1109.727,190.883,-66.168,-179.082,9.264,149.562
C07974=1109.722,191.132,-66.193,-179.080,9.267,149.562
C07975=1109.717,191.380,-66.218,-179.077,9.270,149.562
C07976=1109.713,191.629,-66.243,-179.075,9.272,149.562
C07977=1109.708,191.878,-66.267,-179.073,9.276,149.562
C07978=1109.704,192.127,-66.292,-179.071,9.278,149.562
C07979=1109.699,192.376,-66.316,-179.068,9.281,149.562
C07980=1109.695,192.624,-66.341,-179.066,9.283,149.562
C07981=1109.690,192.873,-66.366,-179.064,9.286,149.562
C07982=1109.686,193.122,-66.390,-179.061,9.290,149.562
C07983=1109.681,193.371,-66.415,-179.060,9.292,149.562
C07984=1109.676,193.619,-66.441,-179.057,9.295,149.562
C07985=1109.673,193.868,-66.465,-179.056,9.298,149.562
C07986=1109.668,194.117,-66.490,-179.053,9.301,149.563
C07987=1109.664,194.365,-66.515,-179.051,9.303,149.563
C07988=1109.659,194.614,-66.540,-179.049,9.306,149.563
C07989=1109.654,194.863,-66.564,-179.046,9.309,149.563
C07990=1109.650,195.111,-66.590,-179.045,9.312,149.563
C07991=1109.645,195.360,-66.614,-179.042,9.315,149.563
C07992=1109.641,195.609,-66.639,-179.040,9.317,149.563
C07993=1109.637,195.857,-66.664,-179.038,9.321,149.563
C07994=1109.632,196.107,-66.689,-179.036,9.323,149.563
C07995=1109.627,196.355,-66.714,-179.034,9.326,149.563
C07996=1109.623,196.604,-66.739,-179.031,9.329,149.563
C07997=1109.618,196.853,-66.764,-179.029,9.333,149.563
C07998=1109.614,197.101,-66.789,-179.026,9.336,149.564
C07999=1109.610,197.350,-66.813,-179.024,9.338,149.564
C08000=1109.605,197.599,-66.839,-179.022,9.341,149.564
C08001=1109.600,197.847,-66.864,-179.019,9.344,149.564
C08002=1109.596,198.096,-66.890,-179.017,9.347,149.564
C08003=1109.592,198.345,-66.914,-179.014,9.350,149.564
C08004=1109.587,198.593,-66.939,-179.011,9.353,149.564
C08005=1109.582,198.842,-66.964,-179.009,9.356,149.564
C08006=1109.579,199.091,-66.989,-179.006,9.359,149.564
C08007=1109.574,199.340,-67.014,-179.003,9.362,149.564
C08008=1109.569,199.588,-67.040,-179.001,9.365,149.564
C08009=1109.565,199.838,-67.065,-178.998,9.368,149.564
C08010=1109.561,200.050,-67.087,-178.996,9.370,149.564
C08011=1109.557,200.263,-67.108,-178.993,9.373,149.564
C08012=1109.554,200.477,-67.130,-178.991,9.376,149.564
C08013=1109.550,200.689,-67.152,-178.989,9.378,149.563
C08014=1109.545,200.903,-67.173,-178.987,9.381,149.564
C08015=1109.542,201.116,-67.195,-178.984,9.383,149.563
C08016=1109.539,201.328,-67.216,-178.982,9.385,149.563
C08017=1109.535,201.542,-67.237,-178.979,9.388,149.563
C08018=1109.531,201.790,-67.263,-178.977,9.391,149.563
C08019=1109.526,202.038,-67.288,-178.974,9.394,149.563
C08020=1109.521,202.288,-67.313,-178.971,9.397,149.563
C08021=1109.517,202.537,-67.339,-178.968,9.400,149.563
C08022=1109.512,202.785,-67.365,-178.966,9.402,149.563
C08023=1109.508,203.034,-67.390,-178.963,9.405,149.563
C08024=1109.503,203.283,-67.415,-178.960,9.408,149.563
C08025=1109.499,203.531,-67.441,-178.957,9.411,149.563
C08026=1109.494,203.780,-67.467,-178.955,9.414,149.563
C08027=1109.491,204.028,-67.492,-178.952,9.417,149.563
C08028=1109.486,204.276,-67.517,-178.949,9.420,149.562
C08029=1109.481,204.526,-67.542,-178.946,9.423,149.563
C08030=1109.477,204.774,-67.567,-178.943,9.425,149.562
C08031=1109.472,205.023,-67.593,-178.940,9.428,149.562
C08032=1109.468,205.272,-67.619,-178.937,9.431,149.562
C08033=1109.463,205.520,-67.644,-178.935,9.434,149.562
C08034=1109.459,205.769,-67.670,-178.932,9.437,149.562
C08035=1109.455,206.017,-67.696,-178.929,9.440,149.562
C08036=1109.451,206.266,-67.722,-178.926,9.442,149.562
C08037=1109.446,206.514,-67.747,-178.923,9.445,149.562
C08038=1109.441,206.764,-67.773,-178.920,9.448,149.562
C08039=1109.436,207.013,-67.798,-178.917,9.452,149.562
C08040=1109.432,207.261,-67.824,-178.914,9.454,149.561
C08041=1109.427,207.510,-67.850,-178.911,9.457,149.561
C08042=1109.423,207.759,-67.875,-178.908,9.460,149.561
C08043=1109.419,208.007,-67.901,-178.906,9.463,149.561
C08044=1109.414,208.255,-67.927,-178.903,9.466,149.561
C08045=1109.410,208.504,-67.953,-178.899,9.470,149.561
C08046=1109.406,208.752,-67.979,-178.896,9.472,149.561
C08047=1109.402,209.001,-68.004,-178.894,9.475,149.561
C08048=1109.397,209.249,-68.030,-178.891,9.478,149.561
C08049=1109.392,209.498,-68.056,-178.888,9.481,149.561
C08050=1109.388,209.747,-68.082,-178.884,9.484,149.561
C08051=1109.383,209.996,-68.108,-178.882,9.487,149.560
C08052=1109.379,210.245,-68.133,-178.879,9.490,149.561
C08053=1109.375,210.492,-68.159,-178.875,9.494,149.560
C08054=1109.370,210.741,-68.185,-178.872,9.497,149.560
C08055=1109.366,210.990,-68.212,-178.870,9.500,149.560
C08056=1109.361,211.239,-68.237,-178.866,9.503,149.560
C08057=1109.357,211.488,-68.263,-178.863,9.506,149.560
C08058=1109.353,211.736,-68.290,-178.861,9.509,149.560
C08059=1109.348,211.984,-68.316,-178.857,9.513,149.560
C08060=1109.343,212.233,-68.341,-178.855,9.516,149.560
C08061=1109.339,212.481,-68.368,-178.851,9.519,149.560
C08062=1109.335,212.730,-68.393,-178.849,9.522,149.560
C08063=1109.330,212.979,-68.420,-178.845,9.526,149.560
C08064=1109.326,213.228,-68.446,-178.843,9.529,149.560
C08065=1109.322,213.476,-68.472,-178.839,9.533,149.560
C08066=1109.318,213.689,-68.494,-178.838,9.535,149.560
C08067=1109.314,213.903,-68.517,-178.836,9.538,149.560
C08068=1109.311,214.115,-68.539,-178.834,9.540,149.560
C08069=1109.307,214.328,-68.562,-178.832,9.542,149.560
C08070=1109.303,214.541,-68.584,-178.830,9.545,149.560
C08071=1109.299,214.754,-68.606,-178.827,9.548,149.560
C08072=1109.295,214.967,-68.629,-178.826,9.550,149.561
C08073=1109.292,215.180,-68.651,-178.824,9.553,149.561
C08074=1109.287,215.429,-68.677,-178.822,9.556,149.561
C08075=1109.283,215.677,-68.704,-178.820,9.558,149.561
C08076=1109.279,215.926,-68.730,-178.817,9.561,149.561
C08077=1109.274,216.174,-68.757,-178.815,9.565,149.561
C08078=1109.270,216.423,-68.783,-178.812,9.568,149.561
C08079=1109.266,216.671,-68.809,-178.811,9.570,149.561
C08080=1109.261,216.921,-68.836,-178.808,9.573,149.561
C08081=1109.256,217.168,-68.862,-178.806,9.577,149.562
C08082=1109.252,217.416,-68.888,-178.803,9.580,149.562
C08083=1109.247,217.665,-68.914,-178.801,9.583,149.562
C08084=1109.244,217.914,-68.941,-178.799,9.585,149.562
C08085=1109.239,218.163,-68.967,-178.797,9.588,149.562
C08086=1109.235,218.411,-68.994,-178.794,9.592,149.562
C08087=1109.230,218.660,-69.020,-178.792,9.595,149.562
C08088=1109.226,218.908,-69.047,-178.789,9.598,149.562
C08089=1109.221,219.157,-69.074,-178.787,9.600,149.562
C08090=1109.217,219.405,-69.099,-178.785,9.604,149.562
C08091=1109.213,219.654,-69.126,-178.783,9.607,149.563
C08092=1109.208,219.902,-69.153,-178.780,9.610,149.563
C08093=1109.203,220.151,-69.179,-178.778,9.613,149.563
C08094=1109.199,220.399,-69.206,-178.775,9.616,149.563
C08095=1109.195,220.648,-69.233,-178.773,9.619,149.563
C08096=1109.191,220.896,-69.259,-178.771,9.622,149.563
C08097=1109.186,221.145,-69.286,-178.769,9.625,149.563
C08098=1109.182,221.393,-69.312,-178.766,9.628,149.563
C08099=1109.178,221.643,-69.339,-178.764,9.632,149.563
C08100=1109.174,221.891,-69.366,-178.761,9.635,149.563
C08101=1109.169,222.140,-69.392,-178.759,9.638,149.563
C08102=1109.165,222.388,-69.419,-178.756,9.641,149.563
C08103=1109.160,222.637,-69.446,-178.755,9.644,149.564
C08104=1109.156,222.885,-69.473,-178.752,9.647,149.564
C08105=1109.152,223.133,-69.499,-178.750,9.650,149.564
C08106=1109.147,223.382,-69.526,-178.747,9.653,149.564
C08107=1109.142,223.631,-69.553,-178.745,9.656,149.564
C08108=1109.138,223.879,-69.579,-178.742,9.659,149.564
C08109=1109.134,224.128,-69.606,-178.739,9.662,149.564
C08110=1109.130,224.376,-69.633,-178.737,9.665,149.564
C08111=1109.125,224.624,-69.660,-178.734,9.668,149.564
C08112=1109.121,224.873,-69.687,-178.733,9.671,149.564
C08113=1109.117,225.122,-69.714,-178.730,9.674,149.564
C08114=1109.112,225.370,-69.741,-178.727,9.677,149.564
C08115=1109.108,225.619,-69.768,-178.725,9.680,149.565
C08116=1109.104,225.867,-69.794,-178.722,9.683,149.564
C08117=1109.099,226.115,-69.821,-178.720,9.686,149.564
C08118=1109.095,226.364,-69.848,-178.717,9.689,149.565
C08119=1109.090,226.612,-69.875,-178.714,9.692,149.565
C08120=1109.087,226.861,-69.902,-178.712,9.695,149.565
C08121=1109.082,227.110,-69.929,-178.709,9.698,149.565
C08122=1109.078,227.323,-69.953,-178.708,9.701,149.565
C08123=1109.074,227.536,-69.975,-178.705,9.703,149.565
C08124=1109.071,227.748,-69.998,-178.703,9.706,149.565
C08125=1109.067,227.961,-70.022,-178.701,9.708,149.565
C08126=1109.063,228.174,-70.045,-178.699,9.710,149.565
C08127=1109.060,228.386,-70.068,-178.696,9.713,149.565
C08128=1109.056,228.599,-70.091,-178.694,9.716,149.565
C08129=1109.052,228.812,-70.115,-178.692,9.718,149.565
C08130=1109.047,229.061,-70.142,-178.689,9.721,149.565
C08131=1109.043,229.309,-70.169,-178.687,9.724,149.565
C08132=1109.039,229.558,-70.195,-178.684,9.727,149.565
C08133=1109.035,229.807,-70.223,-178.681,9.730,149.565
C08134=1109.030,230.055,-70.251,-178.679,9.733,149.565
C08135=1109.026,230.303,-70.278,-178.676,9.735,149.565
C08136=1109.021,230.552,-70.305,-178.673,9.739,149.565
C08137=1109.017,230.801,-70.332,-178.670,9.741,149.565
C08138=1109.012,231.049,-70.359,-178.668,9.743,149.564
C08139=1109.009,231.297,-70.386,-178.665,9.746,149.565
C08140=1109.004,231.545,-70.413,-178.662,9.749,149.564
C08141=1109.000,231.795,-70.441,-178.660,9.752,149.565
C08142=1108.996,232.042,-70.469,-178.657,9.755,149.564
C08143=1108.991,232.291,-70.496,-178.654,9.758,149.564
C08144=1108.986,232.539,-70.523,-178.652,9.760,149.564
C08145=1108.983,232.788,-70.551,-178.649,9.763,149.564
C08146=1108.978,233.037,-70.578,-178.646,9.766,149.564
C08147=1108.973,233.285,-70.605,-178.644,9.769,149.564
C08148=1108.969,233.533,-70.633,-178.641,9.771,149.564
C08149=1108.965,233.782,-70.660,-178.638,9.773,149.564
C08150=1108.960,234.031,-70.687,-178.636,9.777,149.564
C08151=1108.956,234.278,-70.715,-178.633,9.779,149.564
C08152=1108.952,234.528,-70.742,-178.630,9.782,149.564
C08153=1108.948,234.776,-70.770,-178.628,9.784,149.564
C08154=1108.943,235.024,-70.797,-178.625,9.787,149.564
C08155=1108.939,235.273,-70.825,-178.622,9.790,149.564
C08156=1108.934,235.521,-70.853,-178.620,9.792,149.563
C08157=1108.930,235.769,-70.880,-178.617,9.795,149.563
C08158=1108.926,236.018,-70.908,-178.614,9.797,149.563
C08159=1108.922,236.266,-70.935,-178.612,9.800,149.563
C08160=1108.917,236.515,-70.963,-178.609,9.802,149.563
C08161=1108.913,236.763,-70.991,-178.606,9.805,149.563
C08162=1108.909,237.012,-71.018,-178.603,9.808,149.563
C08163=1108.905,237.260,-71.046,-178.601,9.810,149.563
C08164=1108.900,237.509,-71.073,-178.599,9.813,149.563
C08165=1108.896,237.757,-71.101,-178.596,9.816,149.563
C08166=1108.892,238.005,-71.129,-178.593,9.818,149.562
C08167=1108.887,238.254,-71.157,-178.590,9.821,149.562
C08168=1108.882,238.502,-71.184,-178.588,9.824,149.562
C08169=1108.879,238.750,-71.212,-178.585,9.826,149.562
C08170=1108.874,238.999,-71.240,-178.583,9.828,149.562
C08171=1108.870,239.247,-71.268,-178.580,9.831,149.562
C08172=1108.866,239.495,-71.295,-178.578,9.833,149.562
C08173=1108.862,239.745,-71.323,-178.575,9.836,149.562
C08174=1108.857,239.993,-71.351,-178.572,9.839,149.562
C08175=1108.852,240.241,-71.379,-178.569,9.841,149.562
C08176=1108.848,240.490,-71.406,-178.567,9.844,149.562
C08177=1108.844,240.738,-71.434,-178.564,9.847,149.562
C08178=1108.841,240.950,-71.458,-178.562,9.849,149.562
C08179=1108.837,241.163,-71.482,-178.560,9.851,149.562
C08180=1108.833,241.375,-71.506,-178.558,9.853,149.561
C08181=1108.829,241.589,-71.530,-178.556,9.855,149.562
C08182=1108.826,241.801,-71.554,-178.553,9.857,149.561
C08183=1108.822,242.014,-71.578,-178.550,9.860,149.561
C08184=1108.818,242.227,-71.602,-178.548,9.862,149.561
C08185=1108.815,242.440,-71.626,-178.546,9.864,149.561
C08186=1108.810,242.687,-71.653,-178.544,9.868,149.561
C08187=1108.806,242.936,-71.682,-178.541,9.870,149.561
C08188=1108.801,243.184,-71.710,-178.539,9.873,149.561
C08189=1108.798,243.433,-71.738,-178.536,9.875,149.561
C08190=1108.793,243.681,-71.766,-178.534,9.877,149.561
C08191=1108.789,243.930,-71.794,-178.531,9.880,149.561
C08192=1108.784,244.178,-71.822,-178.528,9.883,149.561
C08193=1108.780,244.427,-71.850,-178.526,9.886,149.561
C08194=1108.775,244.675,-71.878,-178.523,9.888,149.561
C08195=1108.772,244.923,-71.906,-178.521,9.891,149.561
C08196=1108.767,245.171,-71.934,-178.519,9.894,149.561
C08197=1108.763,245.420,-71.963,-178.516,9.896,149.561
C08198=1108.759,245.669,-71.991,-178.513,9.900,149.561
C08199=1108.755,245.917,-72.019,-178.511,9.902,149.561
C08200=1108.750,246.166,-72.048,-178.509,9.905,149.561
C08201=1108.746,246.413,-72.075,-178.506,9.908,149.561
C08202=1108.741,246.662,-72.104,-178.503,9.911,149.561
C08203=1108.737,246.910,-72.132,-178.501,9.913,149.561
C08204=1108.733,247.159,-72.160,-178.499,9.916,149.561
C08205=1108.728,247.407,-72.188,-178.496,9.919,149.561
C08206=1108.724,247.656,-72.217,-178.494,9.922,149.561
C08207=1108.720,247.904,-72.246,-178.491,9.925,149.561
C08208=1108.716,248.152,-72.274,-178.488,9.928,149.561
C08209=1108.712,248.400,-72.302,-178.484,9.931,149.561
C08210=1108.707,248.648,-72.330,-178.482,9.934,149.561
C08211=1108.703,248.897,-72.358,-178.479,9.937,149.561
C08212=1108.699,249.146,-72.387,-178.476,9.940,149.561
C08213=1108.695,249.393,-72.416,-178.473,9.943,149.561
C08214=1108.690,249.642,-72.444,-178.470,9.945,149.561
C08215=1108.687,249.891,-72.473,-178.467,9.948,149.560
C08216=1108.681,250.139,-72.501,-178.464,9.951,149.560
C08217=1108.678,250.387,-72.529,-178.461,9.953,149.560
C08218=1108.673,250.635,-72.558,-178.458,9.956,149.560
C08219=1108.669,250.884,-72.586,-178.455,9.958,149.560
C08220=1108.665,251.132,-72.615,-178.452,9.961,149.560
C08221=1108.660,251.380,-72.644,-178.449,9.963,149.559
C08222=1108.656,251.629,-72.672,-178.446,9.966,149.559
C08223=1108.652,251.877,-72.701,-178.443,9.969,149.559
C08224=1108.648,252.125,-72.729,-178.441,9.971,149.559
C08225=1108.643,252.374,-72.758,-178.437,9.973,149.559
C08226=1108.639,252.622,-72.786,-178.435,9.976,149.559
C08227=1108.635,252.870,-72.816,-178.432,9.978,149.558
C08228=1108.630,253.119,-72.844,-178.429,9.981,149.558
C08229=1108.626,253.367,-72.872,-178.427,9.983,149.558
C08230=1108.622,253.615,-72.902,-178.424,9.985,149.558
C08231=1108.618,253.863,-72.930,-178.421,9.988,149.558
C08232=1108.614,254.112,-72.959,-178.418,9.990,149.558
C08233=1108.609,254.360,-72.988,-178.415,9.992,149.558
C08234=1108.606,254.573,-73.012,-178.414,9.995,149.558
C08235=1108.602,254.786,-73.037,-178.411,9.997,149.557
C08236=1108.598,254.997,-73.062,-178.409,9.999,149.557
C08237=1108.594,255.210,-73.087,-178.407,10.001,149.557
C08238=1108.591,255.423,-73.111,-178.405,10.003,149.557
C08239=1108.587,255.636,-73.136,-178.402,10.005,149.557
C08240=1108.584,255.848,-73.160,-178.401,10.007,149.557
C08241=1108.580,256.061,-73.185,-178.398,10.009,149.557
C08242=1108.576,256.309,-73.214,-178.396,10.012,149.557
C08243=1108.572,256.558,-73.243,-178.393,10.014,149.557
C08244=1108.567,256.805,-73.272,-178.390,10.017,149.557
C08245=1108.563,257.054,-73.301,-178.388,10.020,149.557
C08246=1108.559,257.302,-73.329,-178.385,10.023,149.557
C08247=1108.555,257.550,-73.359,-178.382,10.026,149.557
C08248=1108.550,257.799,-73.387,-178.379,10.029,149.557
C08249=1108.546,258.047,-73.416,-178.377,10.032,149.557
C08250=1108.542,258.295,-73.445,-178.374,10.034,149.557
C08251=1108.538,258.544,-73.474,-178.371,10.036,149.557
C08252=1108.533,258.792,-73.504,-178.368,10.039,149.556
C08253=1108.529,259.040,-73.533,-178.366,10.042,149.557
C08254=1108.525,259.288,-73.562,-178.363,10.045,149.556
C08255=1108.521,259.536,-73.590,-178.360,10.048,149.556
C08256=1108.517,259.785,-73.620,-178.357,10.051,149.556
C08257=1108.512,260.033,-73.649,-178.355,10.053,149.556
C08258=1108.508,260.282,-73.678,-178.352,10.056,149.556
C08259=1108.504,260.530,-73.707,-178.349,10.058,149.556
C08260=1108.500,260.778,-73.737,-178.346,10.061,149.556
C08261=1108.495,261.026,-73.766,-178.343,10.064,149.556
C08262=1108.491,261.274,-73.795,-178.340,10.067,149.556
C08263=1108.487,261.522,-73.824,-178.337,10.069,149.556
C08264=1108.483,261.771,-73.853,-178.335,10.071,149.556
C08265=1108.478,262.019,-73.882,-178.332,10.074,149.555
C08266=1108.474,262.268,-73.912,-178.329,10.077,149.555
C08267=1108.470,262.516,-73.941,-178.326,10.080,149.555
C08268=1108.466,262.764,-73.971,-178.323,10.082,149.555
C08269=1108.461,263.012,-74.000,-178.320,10.085,149.555
C08270=1108.457,263.260,-74.029,-178.318,10.088,149.555
C08271=1108.453,263.508,-74.059,-178.315,10.090,149.555
C08272=1108.449,263.757,-74.088,-178.312,10.093,149.555
C08273=1108.444,264.005,-74.118,-178.309,10.095,149.555
C08274=1108.440,264.254,-74.146,-178.306,10.098,149.554
C08275=1108.436,264.502,-74.176,-178.303,10.101,149.554
C08276=1108.432,264.750,-74.205,-178.300,10.103,149.554
C08277=1108.427,264.999,-74.235,-178.298,10.105,149.554
C08278=1108.424,265.246,-74.265,-178.295,10.108,149.554
C08279=1108.419,265.494,-74.294,-178.292,10.111,149.554
C08280=1108.415,265.743,-74.324,-178.289,10.114,149.554
C08281=1108.411,265.991,-74.353,-178.287,10.116,149.554
C08282=1108.407,266.239,-74.383,-178.284,10.118,149.553
C08283=1108.403,266.487,-74.412,-178.281,10.121,149.553
C08284=1108.398,266.736,-74.442,-178.278,10.124,149.553
C08285=1108.394,266.984,-74.471,-178.275,10.126,149.553
C08286=1108.390,267.232,-74.501,-178.272,10.128,149.553
C08287=1108.385,267.480,-74.530,-178.269,10.131,149.553
C08288=1108.381,267.728,-74.560,-178.266,10.134,149.553
C08289=1108.377,267.977,-74.590,-178.263,10.137,149.552
C08290=1108.373,268.189,-74.615,-178.261,10.139,149.552
C08291=1108.370,268.401,-74.640,-178.259,10.141,149.552
C08292=1108.367,268.614,-74.666,-178.257,10.143,149.552
C08293=1108.363,268.826,-74.691,-178.254,10.146,149.552
C08294=1108.359,269.038,-74.717,-178.252,10.148,149.552
C08295=1108.355,269.252,-74.742,-178.249,10.150,149.552
C08296=1108.351,269.464,-74.768,-178.247,10.152,149.552
C08297=1108.348,269.677,-74.794,-178.244,10.154,149.552
C08298=1108.344,269.925,-74.823,-178.242,10.156,149.552
C08299=1108.340,270.172,-74.853,-178.239,10.159,149.552
C08300=1108.336,270.421,-74.883,-178.236,10.162,149.551
C08301=1108.332,270.669,-74.912,-178.233,10.165,149.551
C08302=1108.327,270.918,-74.942,-178.230,10.167,149.551
C08303=1108.323,271.165,-74.972,-178.227,10.170,149.551
C08304=1108.319,271.413,-75.002,-178.225,10.172,149.551
C08305=1108.315,271.661,-75.032,-178.222,10.175,149.551
C08306=1108.310,271.910,-75.062,-178.219,10.178,149.551
C08307=1108.306,272.158,-75.091,-178.216,10.180,149.551
C08308=1108.302,272.406,-75.122,-178.213,10.183,149.550
C08309=1108.298,272.654,-75.151,-178.210,10.186,149.550
C08310=1108.294,272.903,-75.182,-178.207,10.188,149.550
C08311=1108.290,273.151,-75.212,-178.204,10.190,149.550
C08312=1108.286,273.398,-75.242,-178.202,10.193,149.550
C08313=1108.281,273.647,-75.272,-178.199,10.196,149.550
C08314=1108.277,273.895,-75.302,-178.196,10.199,149.550
C08315=1108.273,274.143,-75.331,-178.193,10.201,149.550
C08316=1108.268,274.391,-75.362,-178.190,10.203,149.550
C08317=1108.264,274.640,-75.392,-178.188,10.206,149.550
C08318=1108.261,274.887,-75.422,-178.185,10.209,149.549
C08319=1108.256,275.136,-75.452,-178.182,10.212,149.549
C08320=1108.252,275.384,-75.482,-178.178,10.214,149.549
C08321=1108.248,275.632,-75.512,-178.175,10.217,149.549
C08322=1108.243,275.880,-75.543,-178.172,10.220,149.549
C08323=1108.240,276.128,-75.573,-178.170,10.222,149.549
C08324=1108.236,276.377,-75.603,-178.167,10.224,149.549
C08325=1108.231,276.625,-75.633,-178.164,10.227,149.549
C08326=1108.227,276.872,-75.664,-178.161,10.230,149.548
C08327=1108.222,277.121,-75.694,-178.158,10.232,149.548
C08328=1108.219,277.369,-75.724,-178.155,10.235,149.548
C08329=1108.215,277.617,-75.754,-178.152,10.238,149.548
C08330=1108.210,277.865,-75.784,-178.150,10.240,149.548
C08331=1108.206,278.113,-75.815,-178.147,10.243,149.548
C08332=1108.202,278.362,-75.846,-178.144,10.245,149.547
C08333=1108.198,278.609,-75.876,-178.141,10.248,149.547
C08334=1108.193,278.858,-75.906,-178.138,10.251,149.547
C08335=1108.190,279.105,-75.936,-178.135,10.253,149.547
C08336=1108.186,279.354,-75.967,-178.132,10.256,149.547
C08337=1108.182,279.602,-75.997,-178.129,10.258,149.547
C08338=1108.177,279.850,-76.027,-178.126,10.260,149.547
C08339=1108.173,280.098,-76.058,-178.123,10.263,149.547
C08340=1108.169,280.347,-76.089,-178.120,10.266,149.546
C08341=1108.164,280.595,-76.119,-178.117,10.268,149.546
C08342=1108.160,280.842,-76.150,-178.114,10.271,149.546
C08343=1108.156,281.090,-76.180,-178.111,10.273,149.546
C08344=1108.152,281.339,-76.211,-178.108,10.276,149.546
C08345=1108.148,281.587,-76.242,-178.105,10.278,149.546
C08346=1108.144,281.799,-76.267,-178.103,10.280,149.545
C08347=1108.141,282.011,-76.293,-178.100,10.283,149.545
C08348=1108.137,282.224,-76.320,-178.097,10.285,149.545
C08349=1108.133,282.436,-76.346,-178.095,10.287,149.545
C08350=1108.130,282.648,-76.372,-178.092,10.289,149.545
C08351=1108.126,282.860,-76.398,-178.089,10.291,149.545
C08352=1108.123,283.073,-76.425,-178.087,10.293,149.544
C08353=1108.119,283.286,-76.451,-178.084,10.296,149.544
C08354=1108.115,283.533,-76.482,-178.081,10.299,149.544
C08355=1108.111,283.781,-76.512,-178.079,10.300,149.544
C08356=1108.107,284.030,-76.543,-178.076,10.303,149.544
C08357=1108.102,284.278,-76.574,-178.072,10.305,149.544
C08358=1108.098,284.525,-76.604,-178.069,10.308,149.544
C08359=1108.094,284.774,-76.635,-178.066,10.311,149.543
C08360=1108.090,285.021,-76.667,-178.063,10.313,149.543
C08361=1108.086,285.269,-76.697,-178.060,10.316,149.543
C08362=1108.082,285.518,-76.728,-178.057,10.319,149.543
C08363=1108.078,285.766,-76.759,-178.055,10.321,149.543
C08364=1108.074,286.014,-76.790,-178.051,10.323,149.542
C08365=1108.070,286.262,-76.820,-178.048,10.326,149.542
C08366=1108.065,286.510,-76.851,-178.045,10.329,149.542
C08367=1108.061,286.758,-76.883,-178.042,10.331,149.542
C08368=1108.057,287.006,-76.913,-178.039,10.334,149.542
C08369=1108.054,287.254,-76.944,-178.036,10.336,149.542
C08370=1108.049,287.502,-76.975,-178.033,10.339,149.542
C08371=1108.045,287.750,-77.007,-178.030,10.341,149.541
C08372=1108.041,287.998,-77.037,-178.027,10.343,149.541
C08373=1108.036,288.246,-77.068,-178.024,10.346,149.541
C08374=1108.033,288.495,-77.099,-178.021,10.348,149.541
C08375=1108.028,288.742,-77.130,-178.018,10.351,149.541
C08376=1108.024,288.991,-77.161,-178.015,10.354,149.540
C08377=1108.020,289.238,-77.192,-178.012,10.356,149.540
C08378=1108.016,289.486,-77.224,-178.008,10.359,149.540
C08379=1108.011,289.734,-77.255,-178.006,10.361,149.540
C08380=1108.008,289.982,-77.286,-178.003,10.363,149.540
C08381=1108.004,290.230,-77.317,-178.000,10.366,149.540
C08382=1108.000,290.479,-77.348,-177.997,10.369,149.539
C08383=1107.996,290.726,-77.379,-177.993,10.371,149.539
C08384=1107.992,290.975,-77.410,-177.991,10.374,149.539
C08385=1107.987,291.222,-77.442,-177.987,10.376,149.539
C08386=1107.983,291.471,-77.473,-177.984,10.379,149.539
C08387=1107.979,291.718,-77.504,-177.982,10.381,149.538
C08388=1107.975,291.967,-77.536,-177.979,10.384,149.538
C08389=1107.971,292.214,-77.567,-177.975,10.386,149.538
C08390=1107.967,292.463,-77.598,-177.972,10.389,149.538
C08391=1107.962,292.710,-77.630,-177.969,10.392,149.538
C08392=1107.958,292.959,-77.661,-177.966,10.394,149.538
C08393=1107.954,293.206,-77.692,-177.963,10.397,149.538
C08394=1107.950,293.455,-77.723,-177.960,10.399,149.537
C08395=1107.946,293.703,-77.755,-177.957,10.402,149.537
C08396=1107.942,293.950,-77.787,-177.954,10.404,149.537
C08397=1107.938,294.199,-77.818,-177.951,10.406,149.537
C08398=1107.934,294.446,-77.849,-177.948,10.409,149.537
C08399=1107.930,294.695,-77.880,-177.945,10.412,149.536
C08400=1107.926,294.943,-77.912,-177.942,10.414,149.536
C08401=1107.922,295.190,-77.944,-177.939,10.417,149.536
C08402=1107.916,295.520,-77.985,-177.935,10.420,149.536
C08403=1107.910,295.849,-78.027,-177.931,10.423,149.536
C08404=1107.906,296.178,-78.069,-177.927,10.426,149.535
C08405=1107.900,296.507,-78.111,-177.923,10.430,149.535
C08406=1107.896,296.756,-78.142,-177.920,10.432,149.535
C08407=1107.891,297.003,-78.174,-177.917,10.435,149.535
C08408=1107.888,297.251,-78.206,-177.914,10.438,149.535
C08409=1107.883,297.499,-78.238,-177.910,10.440,149.534
C08410=1107.880,297.747,-78.270,-177.907,10.443,149.534
C08411=1107.876,297.995,-78.301,-177.904,10.445,149.534
C08412=1107.871,298.243,-78.332,-177.901,10.448,149.534
C08413=1107.867,298.491,-78.365,-177.898,10.450,149.534
C08414=1107.863,298.739,-78.397,-177.896,10.452,149.534
C08415=1107.859,298.986,-78.428,-177.892,10.455,149.533
C08416=1107.855,299.235,-78.460,-177.889,10.458,149.533
C08417=1107.851,299.483,-78.492,-177.886,10.460,149.533
C08418=1107.607,288.828,-77.199,-178.016,10.352,149.540
C08419=1107.611,288.579,-77.168,-178.019,10.350,149.541
C08420=1107.615,288.331,-77.138,-178.022,10.348,149.541
C08421=1107.620,288.084,-77.106,-178.025,10.345,149.541
C08422=1107.624,287.835,-77.075,-178.028,10.343,149.541
C08423=1107.628,287.587,-77.045,-178.031,10.340,149.541
C08424=1107.632,287.339,-77.014,-178.034,10.337,149.541
C08425=1107.636,287.091,-76.982,-178.037,10.335,149.542
C08426=1107.640,286.843,-76.951,-178.040,10.332,149.542
C08427=1107.644,286.595,-76.921,-178.043,10.329,149.542
C08428=1107.648,286.347,-76.890,-178.046,10.328,149.542
C08429=1107.652,286.099,-76.859,-178.049,10.325,149.542
C08430=1107.657,285.851,-76.827,-178.052,10.323,149.543
C08431=1107.660,285.603,-76.797,-178.055,10.320,149.543
C08432=1107.665,285.355,-76.766,-178.058,10.317,149.543
C08433=1107.669,285.107,-76.735,-178.061,10.315,149.543
C08434=1107.673,284.858,-76.704,-178.064,10.312,149.543
C08435=1107.677,284.611,-76.674,-178.068,10.309,149.543
C08436=1107.682,284.363,-76.643,-178.071,10.307,149.543
C08437=1107.686,284.114,-76.612,-178.073,10.305,149.544
C08438=1107.690,283.866,-76.582,-178.076,10.302,149.544
C08439=1107.693,283.618,-76.550,-178.079,10.299,149.544
C08440=1107.698,283.370,-76.519,-178.083,10.297,149.544
C08441=1107.702,283.123,-76.489,-178.086,10.294,149.544
C08442=1107.706,282.874,-76.458,-178.089,10.292,149.545
C08443=1107.711,282.553,-76.419,-178.092,10.288,149.545
C08444=1107.717,282.231,-76.379,-178.096,10.285,149.545
C08445=1107.722,281.910,-76.339,-178.100,10.282,149.545
C08446=1107.728,281.589,-76.300,-178.104,10.279,149.545
C08447=1107.732,281.341,-76.269,-178.107,10.276,149.546
C08448=1107.736,281.093,-76.239,-178.110,10.274,149.546
C08449=1107.740,280.844,-76.208,-178.113,10.272,149.546
C08450=1107.745,280.596,-76.178,-178.116,10.269,149.546
C08451=1107.749,280.348,-76.148,-178.119,10.266,149.546
C08452=1107.753,280.100,-76.117,-178.122,10.264,149.546
C08453=1107.757,279.852,-76.086,-178.125,10.261,149.547
C08454=1107.761,279.604,-76.056,-178.127,10.259,149.547
C08455=1107.765,279.356,-76.025,-178.131,10.256,149.547
C08456=1107.770,279.108,-75.995,-178.134,10.254,149.547
C08457=1107.773,278.859,-75.965,-178.137,10.251,149.547
C08458=1107.778,278.611,-75.934,-178.140,10.248,149.547
C08459=1107.782,278.364,-75.904,-178.143,10.246,149.547
C08460=1107.787,278.115,-75.874,-178.146,10.243,149.548
C08461=1107.790,277.867,-75.843,-178.148,10.241,149.548
C08462=1107.795,277.619,-75.812,-178.151,10.238,149.548
C08463=1107.799,277.371,-75.782,-178.154,10.235,149.548
C08464=1107.803,277.123,-75.753,-178.157,10.233,149.548
C08465=1107.807,276.875,-75.722,-178.160,10.230,149.548
C08466=1107.811,276.627,-75.692,-178.163,10.228,149.548
C08467=1107.816,276.378,-75.662,-178.166,10.226,149.548
C08468=1107.819,276.130,-75.631,-178.168,10.223,149.549
C08469=1107.823,275.883,-75.601,-178.171,10.220,149.549
C08470=1107.828,275.634,-75.571,-178.174,10.217,149.549
C08471=1107.831,275.386,-75.541,-178.178,10.215,149.549
C08472=1107.836,275.137,-75.511,-178.181,10.212,149.549
C08473=1107.840,274.890,-75.480,-178.184,10.209,149.549
C08474=1107.844,274.641,-75.451,-178.186,10.207,149.549
C08475=1107.849,274.393,-75.420,-178.189,10.205,149.549
C08476=1107.853,274.146,-75.390,-178.192,10.202,149.550
C08477=1107.857,273.897,-75.360,-178.195,10.199,149.550
C08478=1107.861,273.649,-75.329,-178.198,10.196,149.550
C08479=1107.865,273.401,-75.300,-178.201,10.194,149.550
C08480=1107.869,273.153,-75.270,-178.203,10.192,149.550
C08481=1107.873,272.905,-75.240,-178.206,10.189,149.550
C08482=1107.878,272.656,-75.210,-178.209,10.186,149.550
C08483=1107.882,272.408,-75.180,-178.212,10.184,149.550
C08484=1107.886,272.160,-75.151,-178.215,10.181,149.551
C08485=1107.890,271.911,-75.120,-178.218,10.178,149.551
C08486=1107.895,271.663,-75.090,-178.221,10.175,149.551
C08487=1107.899,271.415,-75.061,-178.223,10.173,149.551
C08488=1107.903,271.167,-75.030,-178.226,10.171,149.551
C08489=1107.907,270.919,-75.001,-178.229,10.168,149.551
C08490=1107.912,270.670,-74.971,-178.232,10.165,149.551
C08491=1107.916,270.423,-74.941,-178.235,10.162,149.551
C08492=1107.920,270.175,-74.911,-178.237,10.160,149.551
C08493=1107.924,269.926,-74.882,-178.240,10.158,149.551
C08494=1107.928,269.679,-74.852,-178.243,10.155,149.552
C08495=1107.931,269.466,-74.826,-178.245,10.153,149.552
C08496=1107.935,269.253,-74.801,-178.248,10.150,149.552
C08497=1107.939,269.041,-74.775,-178.251,10.148,149.552
C08498=1107.942,268.828,-74.750,-178.253,10.146,149.552
C08499=1107.946,268.616,-74.724,-178.255,10.144,149.552
C08500=1107.950,268.404,-74.699,-178.258,10.141,149.552
C08501=1107.953,268.191,-74.674,-178.260,10.139,149.552
C08502=1107.957,267.979,-74.648,-178.262,10.137,149.552
C08503=1107.961,267.731,-74.619,-178.265,10.134,149.552
C08504=1107.966,267.482,-74.589,-178.268,10.131,149.553
C08505=1107.970,267.234,-74.559,-178.272,10.129,149.553
C08506=1107.974,266.986,-74.529,-178.274,10.127,149.553
C08507=1107.978,266.738,-74.500,-178.277,10.124,149.553
C08508=1107.982,266.490,-74.470,-178.280,10.122,149.553
C08509=1107.986,266.241,-74.441,-178.283,10.119,149.553
C08510=1107.991,265.993,-74.411,-178.285,10.117,149.553
C08511=1107.995,265.745,-74.382,-178.288,10.114,149.553
C08512=1107.999,265.497,-74.353,-178.291,10.111,149.554
C08513=1108.003,265.248,-74.323,-178.294,10.109,149.554
C08514=1108.007,265.000,-74.294,-178.296,10.107,149.554
C08515=1108.012,264.752,-74.264,-178.300,10.104,149.554
C08516=1108.016,264.503,-74.235,-178.302,10.101,149.554
C08517=1108.020,264.255,-74.205,-178.305,10.099,149.554
C08518=1108.024,264.007,-74.176,-178.308,10.096,149.554
C08519=1108.029,263.759,-74.147,-178.311,10.094,149.555
C08520=1108.033,263.511,-74.117,-178.314,10.091,149.555
C08521=1108.037,263.263,-74.088,-178.317,10.088,149.555
C08522=1108.041,263.015,-74.058,-178.319,10.086,149.555
C08523=1108.046,262.766,-74.029,-178.322,10.083,149.555
C08524=1108.050,262.518,-73.999,-178.325,10.080,149.555
C08525=1108.054,262.270,-73.970,-178.328,10.078,149.555
C08526=1108.058,262.021,-73.941,-178.331,10.075,149.555
C08527=1108.062,261.773,-73.911,-178.334,10.073,149.555
C08528=1108.067,261.525,-73.883,-178.336,10.070,149.555
C08529=1108.072,261.277,-73.853,-178.339,10.067,149.556
C08530=1108.076,261.028,-73.824,-178.342,10.064,149.556
C08531=1108.080,260.780,-73.794,-178.345,10.062,149.556
C08532=1108.083,260.532,-73.766,-178.348,10.060,149.556
C08533=1108.088,260.283,-73.737,-178.351,10.057,149.556
C08534=1108.092,260.035,-73.707,-178.353,10.054,149.556
C08535=1108.097,259.788,-73.678,-178.356,10.051,149.556
C08536=1108.101,259.539,-73.649,-178.359,10.048,149.556
C08537=1108.106,259.290,-73.620,-178.362,10.045,149.556
C08538=1108.109,259.042,-73.591,-178.364,10.043,149.556
C08539=1108.113,258.794,-73.562,-178.367,10.040,149.556
C08540=1108.117,258.546,-73.532,-178.370,10.038,149.556
C08541=1108.122,258.298,-73.504,-178.373,10.035,149.556
C08542=1108.127,258.049,-73.474,-178.376,10.032,149.557
C08543=1108.130,257.801,-73.446,-178.378,10.029,149.557
C08544=1108.135,257.553,-73.417,-178.381,10.026,149.557
C08545=1108.139,257.304,-73.387,-178.383,10.024,149.557
C08546=1108.144,257.056,-73.359,-178.386,10.021,149.557
C08547=1108.147,256.808,-73.330,-178.389,10.018,149.557
C08548=1108.151,256.560,-73.301,-178.392,10.016,149.557
C08549=1108.156,256.311,-73.272,-178.395,10.013,149.557
C08550=1108.160,256.063,-73.243,-178.397,10.010,149.557
C08551=1108.164,255.850,-73.218,-178.399,10.008,149.557
C08552=1108.168,255.638,-73.194,-178.401,10.005,149.557
C08553=1108.171,255.425,-73.169,-178.404,10.003,149.557
C08554=1108.175,255.213,-73.145,-178.406,10.001,149.557
C08555=1108.178,255.001,-73.120,-178.408,9.999,149.557
C08556=1108.182,254.788,-73.095,-178.410,9.997,149.557
C08557=1108.185,254.575,-73.070,-178.412,9.995,149.557
C08558=1108.189,254.363,-73.046,-178.415,9.993,149.558
C08559=1108.194,254.114,-73.018,-178.418,9.990,149.558
C08560=1108.198,253.866,-72.988,-178.420,9.988,149.558
C08561=1108.202,253.618,-72.960,-178.423,9.986,149.558
C08562=1108.206,253.369,-72.930,-178.426,9.983,149.558
C08563=1108.211,253.121,-72.902,-178.428,9.981,149.558
C08564=1108.215,252.873,-72.873,-178.431,9.978,149.558
C08565=1108.219,252.624,-72.845,-178.433,9.976,149.558
C08566=1108.223,252.376,-72.817,-178.437,9.974,149.559
C08567=1108.228,252.128,-72.787,-178.440,9.971,149.559
C08568=1108.232,251.879,-72.759,-178.442,9.969,149.559
C08569=1108.236,251.631,-72.731,-178.445,9.966,149.559
C08570=1108.241,251.383,-72.701,-178.448,9.964,149.559
C08571=1108.244,251.135,-72.673,-178.451,9.961,149.559
C08572=1108.249,250.886,-72.645,-178.454,9.959,149.560
C08573=1108.253,250.638,-72.616,-178.457,9.956,149.560
C08574=1108.257,250.389,-72.587,-178.460,9.954,149.560
C08575=1108.262,250.142,-72.559,-178.463,9.951,149.560
C08576=1108.266,249.893,-72.531,-178.466,9.949,149.560
C08577=1108.270,249.645,-72.502,-178.469,9.946,149.560
C08578=1108.275,249.397,-72.473,-178.472,9.943,149.560
C08579=1108.278,249.148,-72.445,-178.475,9.940,149.561
C08580=1108.283,248.899,-72.417,-178.478,9.938,149.561
C08581=1108.287,248.651,-72.389,-178.481,9.935,149.561
C08582=1108.292,248.402,-72.360,-178.483,9.932,149.561
C08583=1108.296,248.155,-72.332,-178.486,9.929,149.561
C08584=1108.300,247.906,-72.303,-178.489,9.926,149.561
C08585=1108.304,247.658,-72.275,-178.491,9.923,149.561
C08586=1108.309,247.409,-72.246,-178.494,9.920,149.561
C08587=1108.313,247.161,-72.218,-178.497,9.917,149.561
C08588=1108.317,246.913,-72.190,-178.499,9.914,149.561
C08589=1108.322,246.664,-72.162,-178.502,9.911,149.561
C08590=1108.326,246.416,-72.134,-178.504,9.909,149.561
C08591=1108.331,246.167,-72.105,-178.507,9.906,149.561
C08592=1108.334,245.919,-72.077,-178.509,9.903,149.561
C08593=1108.339,245.671,-72.049,-178.512,9.901,149.561
C08594=1108.343,245.422,-72.021,-178.514,9.898,149.561
C08595=1108.348,245.174,-71.993,-178.517,9.895,149.561
C08596=1108.351,244.926,-71.965,-178.520,9.892,149.561
C08597=1108.356,244.677,-71.936,-178.522,9.889,149.561
C08598=1108.360,244.429,-71.908,-178.524,9.887,149.561
C08599=1108.364,244.181,-71.880,-178.527,9.884,149.561
C08600=1108.369,243.932,-71.852,-178.529,9.882,149.561
C08601=1108.373,243.684,-71.824,-178.532,9.879,149.561
C08602=1108.377,243.436,-71.796,-178.535,9.876,149.561
C08603=1108.382,243.187,-71.767,-178.537,9.873,149.561
C08604=1108.386,242.939,-71.739,-178.540,9.871,149.561
C08605=1108.391,242.690,-71.712,-178.543,9.868,149.561
C08606=1108.394,242.442,-71.684,-178.545,9.865,149.561
C08607=1108.398,242.229,-71.660,-178.547,9.863,149.561
C08608=1108.402,242.016,-71.636,-178.549,9.861,149.561
C08609=1108.406,241.804,-71.611,-178.552,9.859,149.561
C08610=1108.409,241.591,-71.588,-178.554,9.857,149.561
C08611=1108.413,241.378,-71.564,-178.556,9.854,149.561
C08612=1108.417,241.167,-71.540,-178.558,9.852,149.561
C08613=1108.421,240.953,-71.516,-178.561,9.849,149.561
C08614=1108.424,240.741,-71.492,-178.563,9.847,149.562
C08615=1108.428,240.492,-71.465,-178.565,9.845,149.562
C08616=1108.433,240.244,-71.436,-178.568,9.842,149.562
C08617=1108.437,239.995,-71.408,-178.571,9.839,149.562
C08618=1108.441,239.747,-71.381,-178.573,9.837,149.562
C08619=1108.446,239.499,-71.353,-178.576,9.835,149.562
C08620=1108.450,239.250,-71.325,-178.579,9.832,149.562
C08621=1108.454,239.002,-71.297,-178.581,9.830,149.562
C08622=1108.459,238.753,-71.269,-178.584,9.827,149.562
C08623=1108.463,238.505,-71.242,-178.587,9.824,149.562
C08624=1108.467,238.256,-71.214,-178.589,9.822,149.562
C08625=1108.471,238.008,-71.186,-178.592,9.819,149.562
C08626=1108.476,237.760,-71.159,-178.595,9.816,149.562
C08627=1108.480,237.511,-71.131,-178.597,9.813,149.563
C08628=1108.484,237.263,-71.103,-178.600,9.811,149.563
C08629=1108.489,237.014,-71.076,-178.602,9.808,149.563
C08630=1108.493,236.766,-71.048,-178.605,9.806,149.563
C08631=1108.497,236.518,-71.020,-178.608,9.804,149.563
C08632=1108.502,236.269,-70.993,-178.611,9.801,149.563
C08633=1108.506,236.021,-70.965,-178.613,9.798,149.563
C08634=1108.511,235.772,-70.938,-178.615,9.796,149.563
C08635=1108.515,235.523,-70.909,-178.618,9.793,149.563
C08636=1108.519,235.275,-70.882,-178.621,9.790,149.563
C08637=1108.524,235.027,-70.855,-178.624,9.788,149.563
C08638=1108.528,234.778,-70.827,-178.626,9.785,149.563
C08639=1108.532,234.529,-70.800,-178.629,9.782,149.564
C08640=1108.537,234.282,-70.772,-178.632,9.780,149.564
C08641=1108.541,234.032,-70.745,-178.634,9.777,149.564
C08642=1108.545,233.784,-70.717,-178.637,9.775,149.564
C08643=1108.550,233.536,-70.690,-178.640,9.772,149.564
C08644=1108.554,233.288,-70.662,-178.643,9.769,149.564
C08645=1108.558,233.039,-70.635,-178.645,9.767,149.564
C08646=1108.562,232.791,-70.608,-178.648,9.764,149.564
C08647=1108.566,232.543,-70.581,-178.650,9.761,149.564
C08648=1108.570,232.294,-70.553,-178.653,9.758,149.564
C08649=1108.575,232.045,-70.526,-178.656,9.755,149.564
C08650=1108.579,231.797,-70.498,-178.658,9.753,149.564
C08651=1108.584,231.549,-70.471,-178.661,9.750,149.564
C08652=1108.588,231.300,-70.444,-178.664,9.748,149.564
C08653=1108.593,231.051,-70.417,-178.666,9.744,149.564
C08654=1108.597,230.803,-70.389,-178.669,9.742,149.564
C08655=1108.602,230.555,-70.362,-178.672,9.739,149.564
C08656=1108.605,230.306,-70.335,-178.674,9.737,149.565
C08657=1108.610,230.057,-70.308,-178.677,9.734,149.564
C08658=1108.614,229.809,-70.280,-178.680,9.731,149.565
C08659=1108.619,229.561,-70.253,-178.682,9.728,149.564
C08660=1108.623,229.312,-70.226,-178.685,9.725,149.565
C08661=1108.628,229.063,-70.199,-178.688,9.722,149.565
C08662=1108.631,228.815,-70.172,-178.690,9.719,149.564
C08663=1108.635,228.602,-70.149,-178.692,9.717,149.565
C08664=1108.639,228.390,-70.126,-178.694,9.714,149.565
C08665=1108.643,228.177,-70.102,-178.697,9.711,149.565
C08666=1108.646,227.964,-70.079,-178.699,9.709,149.565
C08667=1108.650,227.751,-70.056,-178.701,9.707,149.565
C08668=1108.654,227.539,-70.033,-178.704,9.704,149.565
C08669=1108.658,227.326,-70.009,-178.705,9.702,149.564
C08670=1108.661,227.112,-69.987,-178.707,9.699,149.564
C08671=1108.666,226.864,-69.960,-178.710,9.696,149.565
C08672=1108.670,226.616,-69.932,-178.713,9.693,149.564
C08673=1108.675,226.368,-69.905,-178.715,9.690,149.564
C08674=1108.679,226.119,-69.878,-178.718,9.687,149.564
C08675=1108.683,225.870,-69.851,-178.720,9.684,149.564
C08676=1108.688,225.622,-69.824,-178.723,9.681,149.564
C08677=1108.692,225.373,-69.798,-178.725,9.678,149.564
C08678=1108.696,225.124,-69.771,-178.727,9.675,149.564
C08679=1108.701,224.876,-69.744,-178.730,9.672,149.564
C08680=1108.705,224.628,-69.718,-178.732,9.669,149.564
C08681=1108.710,224.379,-69.691,-178.735,9.666,149.564
C08682=1108.714,224.131,-69.664,-178.737,9.663,149.564
C08683=1108.718,223.882,-69.637,-178.740,9.660,149.564
C08684=1108.722,223.633,-69.610,-178.742,9.657,149.564
C08685=1108.727,223.385,-69.583,-178.745,9.654,149.564
C08686=1108.731,223.137,-69.556,-178.747,9.651,149.564
C08687=1108.736,222.887,-69.530,-178.749,9.648,149.563
C08688=1108.740,222.639,-69.503,-178.752,9.645,149.563
C08689=1108.744,222.391,-69.476,-178.754,9.642,149.563
C08690=1108.749,222.142,-69.449,-178.757,9.639,149.563
C08691=1108.753,221.894,-69.423,-178.759,9.636,149.563
C08692=1108.758,221.646,-69.396,-178.762,9.632,149.563
C08693=1108.762,221.397,-69.370,-178.764,9.629,149.563
C08694=1108.767,221.148,-69.343,-178.766,9.627,149.563
C08695=1108.770,220.900,-69.316,-178.769,9.624,149.563
C08696=1108.775,220.652,-69.289,-178.771,9.621,149.563
C08697=1108.780,220.403,-69.263,-178.774,9.618,149.563
C08698=1108.784,220.154,-69.236,-178.776,9.614,149.563
C08699=1108.789,219.906,-69.209,-178.778,9.611,149.562
C08700=1108.793,219.657,-69.184,-178.781,9.608,149.562
C08701=1108.798,219.409,-69.157,-178.783,9.606,149.562
C08702=1108.801,219.160,-69.130,-178.785,9.602,149.562
C08703=1108.806,218.912,-69.104,-178.788,9.599,149.562
C08704=1108.810,218.663,-69.077,-178.790,9.596,149.562
C08705=1108.814,218.415,-69.051,-178.792,9.593,149.562
C08706=1108.819,218.166,-69.025,-178.794,9.590,149.562
C08707=1108.823,217.918,-68.998,-178.797,9.587,149.562
C08708=1108.828,217.668,-68.972,-178.799,9.584,149.561
C08709=1108.832,217.420,-68.945,-178.801,9.581,149.561
C08710=1108.837,217.171,-68.919,-178.804,9.578,149.561
C08711=1108.841,216.923,-68.892,-178.806,9.575,149.561
C08712=1108.845,216.675,-68.866,-178.808,9.572,149.561
C08713=1108.850,216.426,-68.840,-178.810,9.569,149.561
C08714=1108.854,216.177,-68.813,-178.813,9.566,149.561
C08715=1108.858,215.929,-68.787,-178.815,9.563,149.561
C08716=1108.863,215.680,-68.760,-178.817,9.560,149.561
C08717=1108.867,215.431,-68.735,-178.819,9.557,149.560
C08718=1108.872,215.182,-68.708,-178.822,9.554,149.560
C08719=1108.875,214.970,-68.686,-178.824,9.551,149.560
C08720=1108.879,214.757,-68.664,-178.826,9.549,149.560
C08721=1108.883,214.544,-68.641,-178.828,9.547,149.560
C08722=1108.886,214.331,-68.618,-178.830,9.544,149.560
C08723=1108.890,214.119,-68.596,-178.832,9.541,149.560
C08724=1108.894,213.905,-68.574,-178.834,9.538,149.560
C08725=1108.897,213.692,-68.551,-178.835,9.536,149.560
C08726=1108.902,213.479,-68.528,-178.837,9.534,149.560
C08727=1108.906,213.231,-68.502,-178.840,9.530,149.560
C08728=1108.910,212.982,-68.477,-178.843,9.527,149.560
C08729=1108.914,212.734,-68.450,-178.847,9.523,149.560
C08730=1108.919,212.484,-68.424,-178.850,9.520,149.560
C08731=1108.924,212.236,-68.399,-178.853,9.517,149.560
C08732=1108.928,211.988,-68.372,-178.856,9.514,149.560
C08733=1108.932,211.739,-68.346,-178.859,9.510,149.560
C08734=1108.937,211.490,-68.320,-178.862,9.507,149.560
C08735=1108.941,211.242,-68.293,-178.865,9.504,149.560
C08736=1108.945,210.993,-68.268,-178.868,9.501,149.560
C08737=1108.950,210.745,-68.242,-178.871,9.498,149.560
C08738=1108.954,210.496,-68.217,-178.874,9.495,149.560
C08739=1108.959,210.247,-68.190,-178.877,9.491,149.560
C08740=1108.964,209.998,-68.165,-178.880,9.488,149.560
C08741=1108.967,209.750,-68.138,-178.883,9.486,149.560
C08742=1108.972,209.502,-68.113,-178.886,9.482,149.560
C08743=1108.977,209.253,-68.087,-178.889,9.479,149.560
C08744=1108.981,209.005,-68.061,-178.892,9.476,149.561
C08745=1108.986,208.755,-68.035,-178.895,9.474,149.561
C08746=1108.990,208.507,-68.009,-178.898,9.470,149.561
C08747=1108.995,208.259,-67.984,-178.901,9.467,149.561
C08748=1108.999,208.010,-67.958,-178.904,9.464,149.561
C08749=1109.003,207.761,-67.932,-178.907,9.461,149.561
C08750=1109.007,207.512,-67.906,-178.909,9.458,149.561
C08751=1109.012,207.264,-67.881,-178.913,9.455,149.561
C08752=1109.016,207.015,-67.855,-178.916,9.452,149.561
C08753=1109.021,206.766,-67.830,-178.919,9.449,149.561
C08754=1109.026,206.518,-67.804,-178.921,9.446,149.561
C08755=1109.030,206.269,-67.778,-178.924,9.443,149.562
C08756=1109.034,206.021,-67.753,-178.927,9.441,149.562
C08757=1109.038,205.772,-67.727,-178.930,9.438,149.562
C08758=1109.043,205.524,-67.702,-178.933,9.435,149.562
C08759=1109.047,205.275,-67.676,-178.936,9.432,149.562
C08760=1109.051,205.026,-67.650,-178.939,9.429,149.562
C08761=1109.056,204.778,-67.625,-178.942,9.426,149.562
C08762=1109.061,204.529,-67.599,-178.945,9.423,149.562
C08763=1109.065,204.280,-67.574,-178.948,9.420,149.562
C08764=1109.070,204.032,-67.548,-178.951,9.417,149.562
C08765=1109.074,203.783,-67.523,-178.954,9.414,149.563
C08766=1109.078,203.534,-67.497,-178.956,9.411,149.563
C08767=1109.083,203.286,-67.472,-178.959,9.409,149.563
C08768=1109.088,203.037,-67.447,-178.962,9.406,149.563
C08769=1109.093,202.789,-67.421,-178.964,9.403,149.563
C08770=1109.097,202.540,-67.395,-178.967,9.400,149.563
C08771=1109.101,202.291,-67.370,-178.970,9.397,149.563
C08772=1109.106,202.042,-67.345,-178.972,9.395,149.563
C08773=1109.110,201.794,-67.320,-178.975,9.392,149.563
C08774=1109.114,201.545,-67.294,-178.978,9.389,149.563
C08775=1109.118,201.332,-67.273,-178.981,9.386,149.563
C08776=1109.122,201.119,-67.251,-178.983,9.384,149.563
C08777=1109.125,200.906,-67.229,-178.985,9.382,149.563
C08778=1109.129,200.692,-67.208,-178.987,9.379,149.563
C08779=1109.133,200.480,-67.186,-178.989,9.377,149.563
C08780=1109.137,200.267,-67.164,-178.992,9.374,149.563
C08781=1109.141,200.053,-67.143,-178.994,9.372,149.563
C08782=1109.145,199.841,-67.121,-178.996,9.369,149.563
C08783=1109.149,199.591,-67.096,-178.999,9.366,149.563
C08784=1109.154,199.343,-67.070,-179.002,9.363,149.563
C08785=1109.158,199.094,-67.046,-179.004,9.360,149.563
C08786=1109.163,198.846,-67.021,-179.007,9.358,149.563
C08787=1109.167,198.597,-66.995,-179.010,9.354,149.563
C08788=1109.172,198.348,-66.970,-179.012,9.351,149.563
C08789=1109.176,198.100,-66.945,-179.015,9.348,149.563
C08790=1109.181,197.851,-66.920,-179.017,9.345,149.563
C08791=1109.185,197.602,-66.895,-179.019,9.343,149.563
C08792=1109.189,197.354,-66.871,-179.022,9.340,149.563
C08793=1109.194,197.104,-66.846,-179.024,9.337,149.563
C08794=1109.199,196.856,-66.820,-179.027,9.334,149.563
C08795=1109.203,196.607,-66.795,-179.029,9.331,149.563
C08796=1109.207,196.359,-66.770,-179.032,9.327,149.563
C08797=1109.212,196.110,-66.745,-179.033,9.325,149.563
C08798=1109.217,195.862,-66.720,-179.036,9.322,149.563
C08799=1109.220,195.613,-66.695,-179.039,9.319,149.563
C08800=1109.226,195.364,-66.671,-179.040,9.316,149.563
C08801=1109.230,195.115,-66.645,-179.043,9.313,149.563
C08802=1109.234,194.867,-66.621,-179.044,9.311,149.562
C08803=1109.239,194.617,-66.596,-179.047,9.307,149.562
C08804=1109.243,194.369,-66.571,-179.049,9.305,149.562
C08805=1109.247,194.120,-66.546,-179.051,9.302,149.562
C08806=1109.252,193.871,-66.521,-179.053,9.298,149.562
C08807=1109.256,193.623,-66.496,-179.055,9.296,149.562
C08808=1109.261,193.374,-66.472,-179.058,9.293,149.562
C08809=1109.265,193.126,-66.448,-179.060,9.291,149.562
C08810=1109.270,192.877,-66.422,-179.062,9.288,149.562
C08811=1109.275,192.628,-66.397,-179.064,9.285,149.562
C08812=1109.279,192.379,-66.373,-179.067,9.282,149.562
C08813=1109.284,192.130,-66.348,-179.069,9.279,149.562
C08814=1109.287,191.882,-66.323,-179.071,9.276,149.562
C08815=1109.292,191.633,-66.298,-179.073,9.273,149.561
C08816=1109.297,191.385,-66.274,-179.075,9.271,149.561
C08817=1109.301,191.135,-66.249,-179.078,9.268,149.561
C08818=1109.306,190.887,-66.225,-179.080,9.265,149.561
C08819=1109.311,190.638,-66.200,-179.082,9.262,149.561
C08820=1109.315,190.389,-66.175,-179.085,9.259,149.561
C08821=1109.319,190.141,-66.150,-179.086,9.257,149.561
C08822=1109.324,189.891,-66.125,-179.089,9.254,149.561
C08823=1109.328,189.643,-66.101,-179.091,9.251,149.561
C08824=1109.333,189.395,-66.077,-179.093,9.248,149.561
C08825=1109.337,189.145,-66.052,-179.096,9.245,149.561
C08826=1109.342,188.897,-66.028,-179.098,9.243,149.561
C08827=1109.347,188.648,-66.004,-179.100,9.240,149.561
C08828=1109.351,188.399,-65.979,-179.102,9.237,149.561
C08829=1109.356,188.150,-65.954,-179.105,9.234,149.561
C08830=1109.360,187.902,-65.930,-179.107,9.231,149.561
C08831=1109.364,187.688,-65.909,-179.109,9.229,149.561
C08832=1109.368,187.476,-65.889,-179.111,9.227,149.561
C08833=1109.371,187.262,-65.867,-179.113,9.224,149.561
C08834=1109.375,187.049,-65.845,-179.115,9.222,149.561
C08835=1109.379,186.836,-65.825,-179.117,9.220,149.561
C08836=1109.383,186.623,-65.804,-179.119,9.217,149.561
C08837=1109.387,186.410,-65.783,-179.121,9.214,149.561
C08838=1109.391,186.197,-65.762,-179.123,9.212,149.560
C08839=1109.395,185.948,-65.739,-179.125,9.209,149.560
C08840=1109.400,185.698,-65.714,-179.127,9.206,149.560
C08841=1109.404,185.450,-65.690,-179.130,9.203,149.560
C08842=1109.409,185.201,-65.665,-179.132,9.201,149.560
C08843=1109.414,184.953,-65.641,-179.135,9.198,149.560
C08844=1109.418,184.703,-65.616,-179.137,9.195,149.560
C08845=1109.422,184.455,-65.592,-179.139,9.193,149.560
C08846=1109.427,184.206,-65.568,-179.142,9.190,149.560
C08847=1109.432,183.958,-65.544,-179.144,9.187,149.560
C08848=1109.436,183.708,-65.520,-179.146,9.183,149.560
C08849=1109.441,183.459,-65.495,-179.148,9.181,149.560
C08850=1109.445,183.211,-65.471,-179.151,9.178,149.560
C08851=1109.450,182.963,-65.447,-179.153,9.174,149.560
C08852=1109.453,182.714,-65.423,-179.155,9.172,149.560
C08853=1109.459,182.464,-65.399,-179.158,9.169,149.560
C08854=1109.463,182.216,-65.375,-179.160,9.166,149.560
C08855=1109.468,181.967,-65.351,-179.163,9.163,149.560
C08856=1109.472,181.719,-65.327,-179.165,9.160,149.560
C08857=1109.477,181.469,-65.302,-179.167,9.157,149.560
C08858=1109.481,181.221,-65.278,-179.170,9.154,149.560
C08859=1109.486,180.972,-65.254,-179.172,9.151,149.560
C08860=1109.490,180.723,-65.231,-179.175,9.148,149.560
C08861=1109.495,180.475,-65.207,-179.177,9.145,149.559
C08862=1109.499,180.225,-65.182,-179.179,9.142,149.559
C08863=1109.504,179.976,-65.158,-179.181,9.139,149.559
C08864=1109.508,179.728,-65.134,-179.184,9.136,149.559
C08865=1109.513,179.479,-65.110,-179.186,9.133,149.559
C08866=1109.517,179.230,-65.087,-179.189,9.130,149.559
C08867=1109.522,178.982,-65.063,-179.190,9.127,149.559
C08868=1109.526,178.732,-65.039,-179.193,9.124,149.559
C08869=1109.531,178.483,-65.014,-179.195,9.121,149.559
C08870=1109.535,178.235,-64.990,-179.197,9.118,149.559
C08871=1109.540,177.986,-64.967,-179.199,9.115,149.558
C08872=1109.545,177.738,-64.943,-179.201,9.113,149.558
C08873=1109.549,177.489,-64.919,-179.203,9.109,149.558
C08874=1109.554,177.240,-64.895,-179.206,9.106,149.558
C08875=1109.558,176.990,-64.872,-179.208,9.104,149.558
C08876=1109.562,176.742,-64.847,-179.210,9.100,149.558
C08877=1109.567,176.493,-64.824,-179.212,9.097,149.558
C08878=1109.571,176.245,-64.800,-179.214,9.095,149.558
C08879=1109.576,175.996,-64.777,-179.216,9.091,149.558
C08880=1109.580,175.747,-64.753,-179.219,9.088,149.557
C08881=1109.585,175.498,-64.729,-179.221,9.086,149.557
C08882=1109.590,175.249,-64.706,-179.223,9.082,149.557
C08883=1109.594,175.001,-64.682,-179.225,9.079,149.557
C08884=1109.599,174.752,-64.658,-179.227,9.077,149.557
C08885=1109.603,174.503,-64.634,-179.230,9.074,149.557
C08886=1109.608,174.254,-64.611,-179.232,9.070,149.557
C08887=1109.612,174.040,-64.591,-179.234,9.068,149.557
C08888=1109.616,173.827,-64.570,-179.236,9.066,149.557
C08889=1109.620,173.614,-64.550,-179.237,9.063,149.557
C08890=1109.623,173.401,-64.530,-179.239,9.061,149.557
C08891=1109.628,173.187,-64.509,-179.241,9.058,149.556
C08892=1109.631,172.974,-64.489,-179.243,9.056,149.556
C08893=1109.635,172.761,-64.469,-179.245,9.053,149.556
C08894=1109.639,172.548,-64.450,-179.247,9.050,149.556
C08895=1109.644,172.299,-64.426,-179.249,9.048,149.556
C08896=1109.648,172.050,-64.402,-179.251,9.044,149.556
C08897=1109.653,171.801,-64.379,-179.253,9.041,149.556
C08898=1109.657,171.552,-64.354,-179.255,9.039,149.556
C08899=1109.662,171.304,-64.331,-179.257,9.036,149.556
C08900=1109.667,171.055,-64.308,-179.260,9.032,149.556
C08901=1109.672,170.806,-64.285,-179.262,9.030,149.556
C08902=1109.676,170.557,-64.261,-179.264,9.027,149.555
C08903=1109.680,170.309,-64.238,-179.266,9.023,149.555
C08904=1109.685,170.060,-64.215,-179.268,9.021,149.555
C08905=1109.689,169.810,-64.191,-179.270,9.018,149.555
C08906=1109.694,169.561,-64.168,-179.273,9.015,149.555
C08907=1109.699,169.312,-64.144,-179.275,9.011,149.555
C08908=1109.703,169.063,-64.121,-179.277,9.009,149.555
C08909=1109.708,168.814,-64.098,-179.279,9.006,149.555
C08910=1109.712,168.566,-64.074,-179.281,9.002,149.554
C08911=1109.716,168.317,-64.051,-179.283,9.000,149.554
C08912=1109.721,168.068,-64.028,-179.286,8.997,149.554
C08913=1109.726,167.819,-64.004,-179.288,8.993,149.554
C08914=1109.731,167.570,-63.981,-179.290,8.991,149.554
C08915=1109.735,167.321,-63.958,-179.292,8.987,149.554
C08916=1109.739,167.072,-63.935,-179.294,8.984,149.554
C08917=1109.744,166.823,-63.911,-179.296,8.982,149.554
C08918=1109.749,166.575,-63.888,-179.298,8.978,149.553
C08919=1109.753,166.326,-63.866,-179.301,8.975,149.553
C08920=1109.758,166.077,-63.842,-179.303,8.972,149.553
C08921=1109.763,165.828,-63.819,-179.305,8.970,149.553
C08922=1109.767,165.579,-63.795,-179.307,8.966,149.553
C08923=1109.771,165.330,-63.773,-179.309,8.963,149.553
C08924=1109.776,165.081,-63.749,-179.311,8.961,149.553
C08925=1109.781,164.832,-63.726,-179.313,8.957,149.553
C08926=1109.786,164.584,-63.703,-179.316,8.954,149.553
C08927=1109.790,164.335,-63.680,-179.318,8.951,149.552
C08928=1109.795,164.086,-63.658,-179.320,8.948,149.552
C08929=1109.800,163.837,-63.634,-179.322,8.945,149.552
C08930=1109.804,163.588,-63.611,-179.324,8.942,149.552
C08931=1109.808,163.339,-63.588,-179.327,8.938,149.552
C08932=1109.812,163.090,-63.565,-179.328,8.936,149.552
C08933=1109.818,162.842,-63.542,-179.331,8.933,149.552
C08934=1109.822,162.593,-63.519,-179.333,8.929,149.551
C08935=1109.826,162.343,-63.497,-179.336,8.926,149.551
C08936=1109.831,162.094,-63.474,-179.337,8.923,149.551
C08937=1109.836,161.845,-63.450,-179.340,8.920,149.551
C08938=1109.840,161.597,-63.427,-179.342,8.917,149.551
C08939=1109.845,161.348,-63.404,-179.344,8.913,149.551
C08940=1109.849,161.099,-63.382,-179.346,8.911,149.551
C08941=1109.854,160.850,-63.359,-179.348,8.907,149.550
C08942=1109.858,160.601,-63.336,-179.350,8.904,149.550
C08943=1109.862,160.388,-63.317,-179.352,8.902,149.550
C08944=1109.866,160.175,-63.297,-179.354,8.899,149.550
C08945=1109.870,159.961,-63.278,-179.356,8.896,149.550
C08946=1109.875,159.748,-63.259,-179.358,8.893,149.550
C08947=1109.878,159.534,-63.239,-179.359,8.891,149.550
C08948=1109.882,159.321,-63.219,-179.361,8.888,149.550
C08949=1109.887,159.108,-63.200,-179.363,8.885,149.549
C08950=1109.890,158.895,-63.180,-179.365,8.883,149.549
C08951=1109.895,158.645,-63.158,-179.367,8.879,149.549
C08952=1109.899,158.396,-63.135,-179.369,8.877,149.549
C08953=1109.904,158.148,-63.112,-179.371,8.873,149.549
C08954=1109.908,157.899,-63.090,-179.373,8.870,149.549
C08955=1109.913,157.650,-63.067,-179.376,8.867,149.549
C08956=1109.917,157.400,-63.044,-179.378,8.863,149.548
C08957=1109.922,157.152,-63.021,-179.380,8.860,149.548
C08958=1109.927,156.903,-62.999,-179.382,8.857,149.548
C08959=1109.931,156.653,-62.976,-179.384,8.854,149.548
C08960=1109.936,156.405,-62.954,-179.386,8.850,149.548
C08961=1109.941,156.156,-62.931,-179.388,8.847,149.547
C08962=1109.945,155.907,-62.908,-179.390,8.844,149.547
C08963=1109.950,155.658,-62.887,-179.392,8.840,149.547
C08964=1109.955,155.409,-62.863,-179.394,8.838,149.547
C08965=1109.959,155.160,-62.841,-179.396,8.834,149.547
C08966=1109.964,154.911,-62.819,-179.398,8.831,149.547
C08967=1109.968,154.662,-62.796,-179.401,8.828,149.546
C08968=1109.973,154.413,-62.774,-179.403,8.824,149.546
C08969=1109.978,154.165,-62.751,-179.405,8.821,149.546
C08970=1109.982,153.915,-62.729,-179.407,8.817,149.546
C08971=1109.986,153.667,-62.706,-179.409,8.815,149.546
C08972=1109.992,153.418,-62.684,-179.411,8.811,149.545
C08973=1109.996,153.168,-62.662,-179.413,8.808,149.545
C08974=1110.000,152.920,-62.639,-179.415,8.804,149.545
C08975=1110.006,152.671,-62.617,-179.417,8.801,149.545
C08976=1110.010,152.421,-62.595,-179.419,8.797,149.544
C08977=1110.014,152.173,-62.572,-179.422,8.794,149.544
C08978=1110.019,151.924,-62.550,-179.424,8.791,149.544
C08979=1110.024,151.674,-62.528,-179.426,8.787,149.544
C08980=1110.028,151.426,-62.505,-179.428,8.784,149.544
C08981=1110.033,151.177,-62.483,-179.429,8.781,149.543
C08982=1110.038,150.928,-62.461,-179.431,8.778,149.543
C08983=1110.042,150.679,-62.439,-179.433,8.774,149.543
C08984=1110.046,150.430,-62.416,-179.436,8.771,149.543
C08985=1110.051,150.181,-62.395,-179.438,8.767,149.542
C08986=1110.056,149.932,-62.372,-179.440,8.764,149.542
C08987=1110.061,149.683,-62.350,-179.442,8.760,149.542
C08988=1110.065,149.434,-62.328,-179.444,8.757,149.542
C08989=1110.070,149.186,-62.306,-179.446,8.753,149.541
C08990=1110.075,148.936,-62.283,-179.448,8.750,149.541
C08991=1110.080,148.687,-62.261,-179.450,8.746,149.541
C08992=1110.084,148.438,-62.239,-179.452,8.743,149.541
C08993=1110.089,148.189,-62.218,-179.454,8.739,149.540
C08994=1110.093,147.940,-62.196,-179.456,8.735,149.540
C08995=1110.098,147.691,-62.174,-179.458,8.732,149.540
C08996=1110.103,147.442,-62.151,-179.460,8.728,149.540
C08997=1110.108,147.194,-62.129,-179.462,8.725,149.539
C08998=1110.112,146.944,-62.107,-179.464,8.721,149.539
C08999=1110.116,146.731,-62.089,-179.466,8.719,149.539
C09000=1110.120,146.517,-62.070,-179.468,8.715,149.539
C09001=1110.124,146.305,-62.051,-179.469,8.712,149.538
C09002=1110.128,146.090,-62.032,-179.471,8.709,149.538
C09003=1110.132,145.877,-62.013,-179.473,8.706,149.538
C09004=1110.136,145.663,-61.995,-179.474,8.702,149.538
C09005=1110.140,145.450,-61.975,-179.476,8.700,149.537
C09006=1110.143,145.236,-61.957,-179.478,8.696,149.537
C09007=1110.148,144.988,-61.935,-179.479,8.693,149.537
C09008=1110.153,144.738,-61.913,-179.481,8.690,149.536
C09009=1110.157,144.490,-61.891,-179.483,8.686,149.536
C09010=1110.162,144.241,-61.870,-179.484,8.683,149.536
C09011=1110.167,143.992,-61.847,-179.486,8.680,149.536
C09012=1110.171,143.743,-61.826,-179.488,8.676,149.535
C09013=1110.176,143.493,-61.804,-179.490,8.672,149.535
C09014=1110.181,143.244,-61.783,-179.491,8.669,149.534
C09015=1110.185,142.995,-61.761,-179.493,8.666,149.534
C09016=1110.190,142.746,-61.739,-179.495,8.662,149.534
C09017=1110.194,142.497,-61.717,-179.496,8.659,149.533
C09018=1110.199,142.248,-61.695,-179.498,8.656,149.533
C09019=1110.204,142.000,-61.674,-179.500,8.652,149.533
C09020=1110.208,141.751,-61.652,-179.502,8.648,149.533
C09021=1110.213,141.501,-61.631,-179.503,8.645,149.532
C09022=1110.218,141.252,-61.609,-179.505,8.642,149.532
C09023=1110.223,141.003,-61.587,-179.507,8.638,149.532
C09024=1110.227,140.755,-61.565,-179.508,8.635,149.531
C09025=1110.232,140.505,-61.543,-179.510,8.632,149.531
C09026=1110.237,140.256,-61.522,-179.512,8.628,149.531
C09027=1110.242,140.007,-61.501,-179.513,8.625,149.530
C09028=1110.246,139.758,-61.478,-179.515,8.621,149.530
C09029=1110.251,139.509,-61.457,-179.517,8.618,149.530
C09030=1110.255,139.260,-61.436,-179.519,8.614,149.529
C09031=1110.260,139.011,-61.414,-179.520,8.611,149.529
C09032=1110.265,138.762,-61.393,-179.522,8.608,149.529
C09033=1110.269,138.513,-61.371,-179.524,8.604,149.529
C09034=1110.274,138.264,-61.350,-179.525,8.601,149.528
C09035=1110.279,138.015,-61.328,-179.527,8.597,149.528
C09036=1110.283,137.765,-61.307,-179.529,8.594,149.528
C09037=1110.288,137.517,-61.286,-179.530,8.591,149.527
C09038=1110.292,137.268,-61.264,-179.532,8.587,149.527
C09039=1110.297,137.018,-61.243,-179.534,8.584,149.527
C09040=1110.302,136.770,-61.221,-179.535,8.581,149.526
C09041=1110.307,136.521,-61.199,-179.537,8.577,149.526
C09042=1110.311,136.272,-61.179,-179.540,8.574,149.526
C09043=1110.315,136.023,-61.157,-179.541,8.571,149.525
C09044=1110.321,135.774,-61.136,-179.543,8.567,149.525
C09045=1110.325,135.525,-61.114,-179.545,8.564,149.525
C09046=1110.330,135.275,-61.093,-179.546,8.560,149.524
C09047=1110.334,135.027,-61.072,-179.548,8.557,149.524
C09048=1110.339,134.777,-61.051,-179.550,8.554,149.524
C09049=1110.344,134.529,-61.029,-179.552,8.550,149.524
C09050=1110.349,134.279,-61.008,-179.553,8.547,149.523
C09051=1110.353,134.030,-60.987,-179.555,8.544,149.523
C09052=1110.358,133.781,-60.966,-179.557,8.540,149.523
C09053=1110.363,133.532,-60.944,-179.558,8.537,149.522
C09054=1110.368,133.283,-60.923,-179.560,8.534,149.522
C09055=1110.371,133.069,-60.905,-179.562,8.531,149.522
C09056=1110.375,132.856,-60.886,-179.563,8.528,149.522
C09057=1110.379,132.642,-60.868,-179.564,8.525,149.522
C09058=1110.383,132.429,-60.850,-179.567,8.522,149.521
C09059=1110.388,132.215,-60.832,-179.568,8.519,149.521
C09060=1110.392,132.002,-60.814,-179.569,8.516,149.521
C09061=1110.395,131.787,-60.796,-179.570,8.513,149.520
C09062=1110.399,131.574,-60.778,-179.572,8.511,149.520
C09063=1110.404,131.326,-60.756,-179.574,8.507,149.520
C09064=1110.409,131.076,-60.735,-179.576,8.504,149.520
C09065=1110.414,130.827,-60.715,-179.577,8.501,149.519
C09066=1110.418,130.578,-60.693,-179.579,8.497,149.519
C09067=1110.422,130.329,-60.672,-179.581,8.494,149.519
C09068=1110.428,130.080,-60.651,-179.583,8.491,149.519
C09069=1110.432,129.831,-60.630,-179.585,8.487,149.518
C09070=1110.437,129.582,-60.609,-179.586,8.483,149.518
C09071=1110.442,129.333,-60.588,-179.588,8.481,149.518
C09072=1110.447,129.083,-60.567,-179.590,8.477,149.517
C09073=1110.451,128.835,-60.546,-179.592,8.474,149.517
C09074=1110.456,128.585,-60.525,-179.593,8.471,149.517
C09075=1110.460,128.337,-60.505,-179.595,8.467,149.517
C09076=1110.466,128.087,-60.484,-179.597,8.464,149.516
C09077=1110.470,127.839,-60.462,-179.598,8.461,149.516
C09078=1110.475,127.590,-60.442,-179.600,8.457,149.516
C09079=1110.479,127.340,-60.420,-179.602,8.454,149.515
C09080=1110.484,127.091,-60.400,-179.604,8.451,149.515
C09081=1110.489,126.841,-60.379,-179.606,8.447,149.515
C09082=1110.493,126.593,-60.358,-179.607,8.444,149.515
C09083=1110.498,126.344,-60.337,-179.609,8.441,149.514
C09084=1110.503,126.095,-60.316,-179.611,8.437,149.514
C09085=1110.508,125.846,-60.295,-179.613,8.434,149.514
C09086=1110.512,125.597,-60.275,-179.614,8.431,149.513
C09087=1110.517,125.348,-60.255,-179.616,8.427,149.513
C09088=1110.521,125.098,-60.233,-179.618,8.424,149.513
C09089=1110.526,124.849,-60.213,-179.619,8.421,149.513
C09090=1110.531,124.600,-60.192,-179.621,8.417,149.512
C09091=1110.535,124.351,-60.171,-179.623,8.414,149.512
C09092=1110.540,124.102,-60.150,-179.625,8.410,149.512
C09093=1110.545,123.853,-60.130,-179.627,8.407,149.512
C09094=1110.550,123.604,-60.109,-179.628,8.404,149.511
C09095=1110.554,123.355,-60.088,-179.630,8.400,149.511
C09096=1110.559,123.106,-60.068,-179.632,8.397,149.511
C09097=1110.564,122.857,-60.047,-179.634,8.394,149.510
C09098=1110.568,122.608,-60.027,-179.636,8.390,149.510
C09099=1110.574,122.358,-60.006,-179.637,8.387,149.510
C09100=1110.578,122.110,-59.985,-179.639,8.384,149.510
C09101=1110.582,121.861,-59.965,-179.641,8.380,149.509
C09102=1110.588,121.611,-59.944,-179.642,8.378,149.509
C09103=1110.592,121.362,-59.924,-179.644,8.374,149.509
C09104=1110.597,121.113,-59.904,-179.646,8.370,149.508
C09105=1110.602,120.864,-59.883,-179.648,8.367,149.508
C09106=1110.606,120.615,-59.863,-179.650,8.364,149.508
C09107=1110.611,120.366,-59.842,-179.651,8.360,149.508
C09108=1110.616,120.116,-59.821,-179.653,8.357,149.507
C09109=1110.621,119.867,-59.801,-179.655,8.354,149.507
C09110=1110.625,119.618,-59.780,-179.656,8.350,149.507
C09111=1110.629,119.405,-59.763,-179.658,8.347,149.506
C09112=1110.633,119.191,-59.746,-179.659,8.345,149.506
C09113=1110.638,118.977,-59.728,-179.661,8.341,149.506
C09114=1110.641,118.763,-59.710,-179.663,8.338,149.506
C09115=1110.645,118.549,-59.692,-179.664,8.336,149.506
C09116=1110.650,118.336,-59.675,-179.666,8.333,149.505
C09117=1110.653,118.122,-59.658,-179.667,8.330,149.505
C09118=1110.657,117.908,-59.641,-179.668,8.327,149.505
C09119=1110.662,117.659,-59.620,-179.670,8.324,149.504
C09120=1110.667,117.410,-59.599,-179.672,8.320,149.504
C09121=1110.672,117.161,-59.580,-179.674,8.317,149.504
C09122=1110.676,116.912,-59.559,-179.676,8.314,149.504
C09123=1110.681,116.663,-59.539,-179.677,8.310,149.503
C09124=1110.686,116.414,-59.518,-179.679,8.306,149.503
C09125=1110.691,116.165,-59.499,-179.681,8.303,149.503
C09126=1110.695,115.916,-59.478,-179.682,8.300,149.502
C09127=1110.700,115.667,-59.458,-179.684,8.296,149.502
C09128=1110.705,115.417,-59.438,-179.687,8.293,149.502
C09129=1110.710,115.168,-59.417,-179.688,8.290,149.502
C09130=1110.714,114.919,-59.397,-179.690,8.286,149.501
C09131=1110.719,114.669,-59.377,-179.692,8.283,149.501
C09132=1110.723,114.420,-59.357,-179.694,8.279,149.501
C09133=1110.729,114.172,-59.337,-179.695,8.276,149.500
C09134=1110.733,113.923,-59.317,-179.697,8.273,149.500
C09135=1110.738,113.673,-59.296,-179.699,8.269,149.500
C09136=1110.743,113.424,-59.277,-179.700,8.265,149.500
C09137=1110.748,113.175,-59.256,-179.702,8.263,149.499
C09138=1110.752,112.925,-59.237,-179.704,8.259,149.499
C09139=1110.757,112.676,-59.216,-179.706,8.255,149.499
